ABB RAPID module: P810.mod

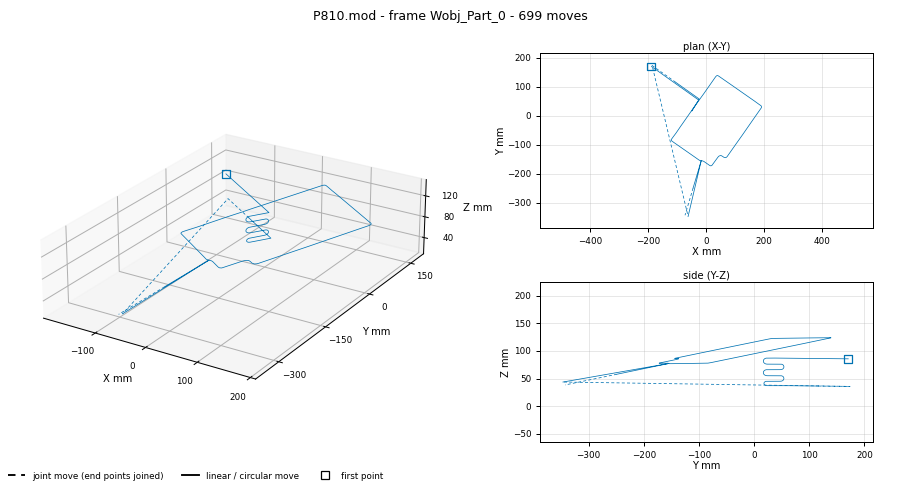
[picture p0: tool path of P810.mod in frame Wobj_Part_0, 699 of 709 moves have a stored position in this frame; points joined in program order, loops and branches not executed]
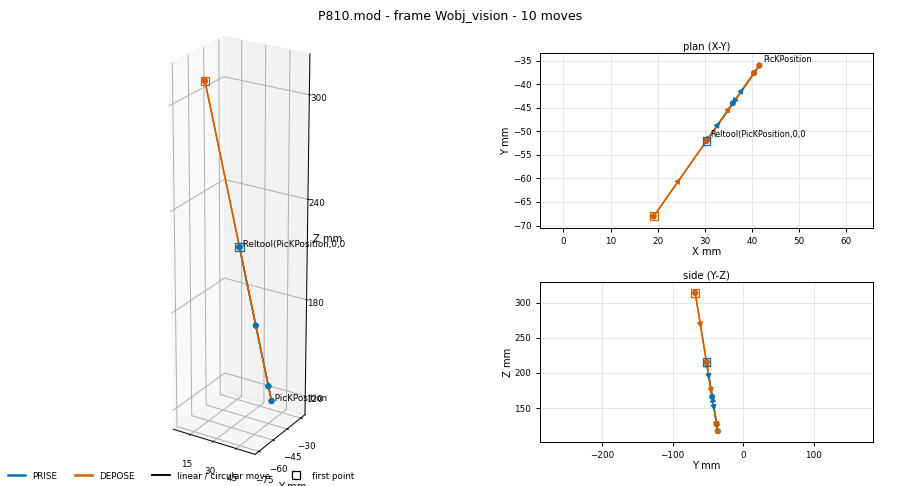
[picture p1: tool path of P810.mod in frame Wobj_vision, 10 of 709 moves have a stored position in this frame; points joined in program order, loops and branches not executed]
MODULE P810

    ! Nom         :P810
    ! Description :
    ! Créé le     :31/05/2023 17:09:28

    LOCAL CONST SPEEDDATA VitesseLente :=[3,500,0,0];
	LOCAL CONST SPEEDDATA VitesseRapide :=[30,500,0,0];
	LOCAL CONST SPEEDDATA VitesseTronconnage :=[2,500,0,0];
	LOCAL CONST SPEEDDATA VitesseTronconnageApp :=[10,500,0,0];
    !
    !Point de prise
    LOCAL PERS Robtarget PicKPosition := [[41.5753348613417,-36.0457521301925,117.430293654676],[0.0866528508359123,-0.450908798340459,0.887153744459286,0.0461602936844953],[0,0,0,0],[8.999999E+09,8.999999E+09,8.999999E+09,8.999999E+09,8.999999E+09,8.999999E+09]];
	LOCAL PERS Pose Ref := [[0,0,0],[1,0,0,0]];
    !
    !Declaration des points de meulage

    !Tr_meulage_motif_1 : Meulage d'un motif
    LOCAL CONST Robtarget Tr_meulage_motif_1_0 := [[-24.86866015625,54.7369140625,87.0190703125],[0.325394831809823,-0.323189731818736,0.626217671016949,-0.630490308557156],[0,0,0,0],[8.999999E+09,8.999999E+09,8.999999E+09,8.999999E+09,8.999999E+09,8.999999E+09]];
    LOCAL CONST Robtarget Tr_meulage_motif_1_1 := [[-25.40796484375,53.8948046875,87.019078125],[0.325394831809823,-0.323189731818736,0.626217671016949,-0.630490308557156],[0,0,0,0],[8.999999E+09,8.999999E+09,8.999999E+09,8.999999E+09,8.999999E+09,8.999999E+09]];
    LOCAL CONST Robtarget Tr_meulage_motif_1_2 := [[-25.94726953125,53.0526953125,87.0190859375],[0.325394831809823,-0.323189731818736,0.626217671016949,-0.630490308557156],[0,0,0,0],[8.999999E+09,8.999999E+09,8.999999E+09,8.999999E+09,8.999999E+09,8.999999E+09]];
    LOCAL CONST Robtarget Tr_meulage_motif_1_3 := [[-26.48657421875,52.2105859375,87.01909375],[0.325394831809823,-0.323189731818736,0.626217671016949,-0.630490308557156],[0,0,0,0],[8.999999E+09,8.999999E+09,8.999999E+09,8.999999E+09,8.999999E+09,8.999999E+09]];
    LOCAL CONST Robtarget Tr_meulage_motif_1_4 := [[-27.025880859375,51.36847265625,87.01909375],[0.325394831809823,-0.323189731818736,0.626217671016949,-0.630490308557156],[0,0,0,0],[8.999999E+09,8.999999E+09,8.999999E+09,8.999999E+09,8.999999E+09,8.999999E+09]];
    LOCAL CONST Robtarget Tr_meulage_motif_1_5 := [[-27.565185546875,50.52636328125,87.0191015625],[0.325394831809823,-0.323189731818736,0.626217671016949,-0.630490308557156],[0,0,0,0],[8.999999E+09,8.999999E+09,8.999999E+09,8.999999E+09,8.999999E+09,8.999999E+09]];
    LOCAL CONST Robtarget Tr_meulage_motif_1_6 := [[-28.104490234375,49.68425390625,87.019109375],[0.325394831809823,-0.323189731818736,0.626217671016949,-0.630490308557156],[0,0,0,0],[8.999999E+09,8.999999E+09,8.999999E+09,8.999999E+09,8.999999E+09,8.999999E+09]];
    LOCAL CONST Robtarget Tr_meulage_motif_1_7 := [[-28.643794921875,48.842140625,87.0191171875],[0.325394831809823,-0.323189731818736,0.626217671016949,-0.630490308557156],[0,0,0,0],[8.999999E+09,8.999999E+09,8.999999E+09,8.999999E+09,8.999999E+09,8.999999E+09]];
    LOCAL CONST Robtarget Tr_meulage_motif_1_8 := [[-29.183099609375,48.00003125,87.019125],[0.325394831809823,-0.323189731818736,0.626217671016949,-0.630490308557156],[0,0,0,0],[8.999999E+09,8.999999E+09,8.999999E+09,8.999999E+09,8.999999E+09,8.999999E+09]];
    LOCAL CONST Robtarget Tr_meulage_motif_1_9 := [[-29.722404296875,47.157921875,87.019125],[0.325394831809823,-0.323189731818736,0.626217671016949,-0.630490308557156],[0,0,0,0],[8.999999E+09,8.999999E+09,8.999999E+09,8.999999E+09,8.999999E+09,8.999999E+09]];
    LOCAL CONST Robtarget Tr_meulage_motif_1_10 := [[-30.2617109375,46.3158125,87.0191328125],[0.325394831809823,-0.323189731818736,0.626217671016949,-0.630490308557156],[0,0,0,0],[8.999999E+09,8.999999E+09,8.999999E+09,8.999999E+09,8.999999E+09,8.999999E+09]];
    LOCAL CONST Robtarget Tr_meulage_motif_1_11 := [[-30.801015625,45.47369921875,87.019140625],[0.325394831809823,-0.323189731818736,0.626217671016949,-0.630490308557156],[0,0,0,0],[8.999999E+09,8.999999E+09,8.999999E+09,8.999999E+09,8.999999E+09,8.999999E+09]];
    LOCAL CONST Robtarget Tr_meulage_motif_1_12 := [[-31.3403203125,44.63158984375,87.0191484375],[0.325394831809823,-0.323189731818736,0.626217671016949,-0.630490308557156],[0,0,0,0],[8.999999E+09,8.999999E+09,8.999999E+09,8.999999E+09,8.999999E+09,8.999999E+09]];
    LOCAL CONST Robtarget Tr_meulage_motif_1_13 := [[-31.879625,43.78948046875,87.01915625],[0.325394831809823,-0.323189731818736,0.626217671016949,-0.630490308557156],[0,0,0,0],[8.999999E+09,8.999999E+09,8.999999E+09,8.999999E+09,8.999999E+09,8.999999E+09]];
    LOCAL CONST Robtarget Tr_meulage_motif_1_14 := [[-32.4189296875,42.9473671875,87.01915625],[0.325394831809823,-0.323189731818736,0.626217671016949,-0.630490308557156],[0,0,0,0],[8.999999E+09,8.999999E+09,8.999999E+09,8.999999E+09,8.999999E+09,8.999999E+09]];
    LOCAL CONST Robtarget Tr_meulage_motif_1_15 := [[-32.958234375,42.1052578125,87.0191640625],[0.325394831809823,-0.323189731818736,0.626217671016949,-0.630490308557156],[0,0,0,0],[8.999999E+09,8.999999E+09,8.999999E+09,8.999999E+09,8.999999E+09,8.999999E+09]];
    LOCAL CONST Robtarget Tr_meulage_motif_1_16 := [[-33.4975390625,41.2631484375,87.019171875],[0.325394831809823,-0.323189731818736,0.626217671016949,-0.630490308557156],[0,0,0,0],[8.999999E+09,8.999999E+09,8.999999E+09,8.999999E+09,8.999999E+09,8.999999E+09]];
    LOCAL CONST Robtarget Tr_meulage_motif_1_17 := [[-34.03684375,40.42103515625,87.0191796875],[0.325394831809823,-0.323189731818736,0.626217671016949,-0.630490308557156],[0,0,0,0],[8.999999E+09,8.999999E+09,8.999999E+09,8.999999E+09,8.999999E+09,8.999999E+09]];
    LOCAL CONST Robtarget Tr_meulage_motif_1_18 := [[-34.5761484375,39.57892578125,87.0191875],[0.325394831809823,-0.323189731818736,0.626217671016949,-0.630490308557156],[0,0,0,0],[8.999999E+09,8.999999E+09,8.999999E+09,8.999999E+09,8.999999E+09,8.999999E+09]];
    LOCAL CONST Robtarget Tr_meulage_motif_1_19 := [[-35.11545703125,38.73681640625,87.0191875],[0.325394831809823,-0.323189731818736,0.626217671016949,-0.630490308557156],[0,0,0,0],[8.999999E+09,8.999999E+09,8.999999E+09,8.999999E+09,8.999999E+09,8.999999E+09]];
    LOCAL CONST Robtarget Tr_meulage_motif_1_20 := [[-35.65476171875,37.89470703125,87.0191953125],[0.325394831809823,-0.323189731818736,0.626217671016949,-0.630490308557156],[0,0,0,0],[8.999999E+09,8.999999E+09,8.999999E+09,8.999999E+09,8.999999E+09,8.999999E+09]];
    LOCAL CONST Robtarget Tr_meulage_motif_1_21 := [[-36.19406640625,37.05259375,87.019203125],[0.325394831809823,-0.323189731818736,0.626217671016949,-0.630490308557156],[0,0,0,0],[8.999999E+09,8.999999E+09,8.999999E+09,8.999999E+09,8.999999E+09,8.999999E+09]];
    LOCAL CONST Robtarget Tr_meulage_motif_1_22 := [[-36.73337109375,36.210484375,87.0192109375],[0.325394831809823,-0.323189731818736,0.626217671016949,-0.630490308557156],[0,0,0,0],[8.999999E+09,8.999999E+09,8.999999E+09,8.999999E+09,8.999999E+09,8.999999E+09]];
    LOCAL CONST Robtarget Tr_meulage_motif_1_23 := [[-37.27267578125,35.368375,87.01921875],[0.325394831809823,-0.323189731818736,0.626217671016949,-0.630490308557156],[0,0,0,0],[8.999999E+09,8.999999E+09,8.999999E+09,8.999999E+09,8.999999E+09,8.999999E+09]];
    LOCAL CONST Robtarget Tr_meulage_motif_1_24 := [[-37.81198046875,34.52626171875,87.0192265625],[0.325394831809823,-0.323189731818736,0.626217671016949,-0.630490308557156],[0,0,0,0],[8.999999E+09,8.999999E+09,8.999999E+09,8.999999E+09,8.999999E+09,8.999999E+09]];
    LOCAL CONST Robtarget Tr_meulage_motif_1_25 := [[-38.35128515625,33.68415234375,87.0192265625],[0.325394831809823,-0.323189731818736,0.626217671016949,-0.630490308557156],[0,0,0,0],[8.999999E+09,8.999999E+09,8.999999E+09,8.999999E+09,8.999999E+09,8.999999E+09]];
    LOCAL CONST Robtarget Tr_meulage_motif_1_26 := [[-38.89058984375,32.84204296875,87.019234375],[0.325394831809823,-0.323189731818736,0.626217671016949,-0.630490308557156],[0,0,0,0],[8.999999E+09,8.999999E+09,8.999999E+09,8.999999E+09,8.999999E+09,8.999999E+09]];
    LOCAL CONST Robtarget Tr_meulage_motif_1_27 := [[-39.42989453125,31.999931640625,87.0192421875],[0.325394831809823,-0.323189731818736,0.626217671016949,-0.630490308557156],[0,0,0,0],[8.999999E+09,8.999999E+09,8.999999E+09,8.999999E+09,8.999999E+09,8.999999E+09]];
    LOCAL CONST Robtarget Tr_meulage_motif_1_28 := [[-39.96919921875,31.157822265625,87.01925],[0.325394831809823,-0.323189731818736,0.626217671016949,-0.630490308557156],[0,0,0,0],[8.999999E+09,8.999999E+09,8.999999E+09,8.999999E+09,8.999999E+09,8.999999E+09]];
    LOCAL CONST Robtarget Tr_meulage_motif_1_29 := [[-40.50850390625,30.3157109375,87.0192578125],[0.325394831809823,-0.323189731818736,0.626217671016949,-0.630490308557156],[0,0,0,0],[8.999999E+09,8.999999E+09,8.999999E+09,8.999999E+09,8.999999E+09,8.999999E+09]];
    LOCAL CONST Robtarget Tr_meulage_motif_1_30 := [[-41.04780859375,29.473599609375,87.0192578125],[0.325394831809823,-0.323189731818736,0.626217671016949,-0.630490308557156],[0,0,0,0],[8.999999E+09,8.999999E+09,8.999999E+09,8.999999E+09,8.999999E+09,8.999999E+09]];
    LOCAL CONST Robtarget Tr_meulage_motif_1_31 := [[-41.58711328125,28.631490234375,87.019265625],[0.325394831809823,-0.323189731818736,0.626217671016949,-0.630490308557156],[0,0,0,0],[8.999999E+09,8.999999E+09,8.999999E+09,8.999999E+09,8.999999E+09,8.999999E+09]];
    LOCAL CONST Robtarget Tr_meulage_motif_1_32 := [[-42.126421875,27.78937890625,87.0192734375],[0.325394831809823,-0.323189731818736,0.626217671016949,-0.630490308557156],[0,0,0,0],[8.999999E+09,8.999999E+09,8.999999E+09,8.999999E+09,8.999999E+09,8.999999E+09]];
    LOCAL CONST Robtarget Tr_meulage_motif_1_33 := [[-42.6657265625,26.94726953125,87.01928125],[0.325394831809823,-0.323189731818736,0.626217671016949,-0.630490308557156],[0,0,0,0],[8.999999E+09,8.999999E+09,8.999999E+09,8.999999E+09,8.999999E+09,8.999999E+09]];
    LOCAL CONST Robtarget Tr_meulage_motif_1_34 := [[-43.20503125,26.105158203125,87.0192890625],[0.325394831809823,-0.323189731818736,0.626217671016949,-0.630490308557156],[0,0,0,0],[8.999999E+09,8.999999E+09,8.999999E+09,8.999999E+09,8.999999E+09,8.999999E+09]];
    LOCAL CONST Robtarget Tr_meulage_motif_1_35 := [[-43.7443359375,25.263046875,87.0192890625],[0.325394831809823,-0.323189731818736,0.626217671016949,-0.630490308557156],[0,0,0,0],[8.999999E+09,8.999999E+09,8.999999E+09,8.999999E+09,8.999999E+09,8.999999E+09]];
    LOCAL CONST Robtarget Tr_meulage_motif_1_36 := [[-44.283640625,24.4209375,87.019296875],[0.325394831809823,-0.323189731818736,0.626217671016949,-0.630490308557156],[0,0,0,0],[8.999999E+09,8.999999E+09,8.999999E+09,8.999999E+09,8.999999E+09,8.999999E+09]];
    LOCAL CONST Robtarget Tr_meulage_motif_1_37 := [[-44.8229453125,23.578826171875,87.0193046875],[0.325394831809823,-0.323189731818736,0.626217671016949,-0.630490308557156],[0,0,0,0],[8.999999E+09,8.999999E+09,8.999999E+09,8.999999E+09,8.999999E+09,8.999999E+09]];
    LOCAL CONST Robtarget Tr_meulage_motif_1_38 := [[-45.36225,22.736716796875,87.0193125],[0.325394831809823,-0.323189731818736,0.626217671016949,-0.630490308557156],[0,0,0,0],[8.999999E+09,8.999999E+09,8.999999E+09,8.999999E+09,8.999999E+09,8.999999E+09]];
    LOCAL CONST Robtarget Tr_meulage_motif_1_39 := [[-45.8972109375,21.90065625,86.9087265625],[0.325394831809823,-0.323189731818736,0.626217671016949,-0.630490308557156],[0,0,0,0],[8.999999E+09,8.999999E+09,8.999999E+09,8.999999E+09,8.999999E+09,8.999999E+09]];
    LOCAL CONST Robtarget Tr_meulage_motif_1_40 := [[-46.40703125,21.10319140625,86.697546875],[0.325394831809823,-0.323189731818736,0.626217671016949,-0.630490308557156],[0,0,0,0],[8.999999E+09,8.999999E+09,8.999999E+09,8.999999E+09,8.999999E+09,8.999999E+09]];
    LOCAL CONST Robtarget Tr_meulage_motif_1_41 := [[-46.86609375,20.384583984375,86.4257109375],[0.325394831809823,-0.323189731818736,0.626217671016949,-0.630490308557156],[0,0,0,0],[8.999999E+09,8.999999E+09,8.999999E+09,8.999999E+09,8.999999E+09,8.999999E+09]];
    LOCAL CONST Robtarget Tr_meulage_motif_1_42 := [[-47.2697109375,19.7525234375,86.1497734375],[0.325394831809823,-0.323189731818736,0.626217671016949,-0.630490308557156],[0,0,0,0],[8.999999E+09,8.999999E+09,8.999999E+09,8.999999E+09,8.999999E+09,8.999999E+09]];
    LOCAL CONST Robtarget Tr_meulage_motif_1_43 := [[-47.861671875,18.824119140625,85.5336640625],[0.325394831809823,-0.323189731818736,0.626217671016949,-0.630490308557156],[0,0,0,0],[8.999999E+09,8.999999E+09,8.999999E+09,8.999999E+09,8.999999E+09,8.999999E+09]];
    LOCAL CONST Robtarget Tr_meulage_motif_1_44 := [[-48.41131640625,17.960271484375,84.686015625],[0.325394831809823,-0.323189731818736,0.626217671016949,-0.630490308557156],[0,0,0,0],[8.999999E+09,8.999999E+09,8.999999E+09,8.999999E+09,8.999999E+09,8.999999E+09]];
    LOCAL CONST Robtarget Tr_meulage_motif_1_45 := [[-48.865390625,17.244478515625,83.66215625],[0.325394831809823,-0.323189731818736,0.626217671016949,-0.630490308557156],[0,0,0,0],[8.999999E+09,8.999999E+09,8.999999E+09,8.999999E+09,8.999999E+09,8.999999E+09]];
    LOCAL CONST Robtarget Tr_meulage_motif_1_46 := [[-49.1253125,16.83124609375,82.5459765625],[0.325394831809823,-0.323189731818736,0.626217671016949,-0.630490308557156],[0,0,0,0],[8.999999E+09,8.999999E+09,8.999999E+09,8.999999E+09,8.999999E+09,8.999999E+09]];
    LOCAL CONST Robtarget Tr_meulage_motif_1_47 := [[-49.13782421875,16.807115234375,81.850015625],[0.325394831809823,-0.323189731818736,0.626217671016949,-0.630490308557156],[0,0,0,0],[8.999999E+09,8.999999E+09,8.999999E+09,8.999999E+09,8.999999E+09,8.999999E+09]];
    LOCAL CONST Robtarget Tr_meulage_motif_1_48 := [[-49.13583984375,16.805841796875,81.188765625],[0.325394831809823,-0.323189731818736,0.626217671016949,-0.630490308557156],[0,0,0,0],[8.999999E+09,8.999999E+09,8.999999E+09,8.999999E+09,8.999999E+09,8.999999E+09]];
    LOCAL CONST Robtarget Tr_meulage_motif_1_49 := [[-49.104265625,16.850779296875,80.5276796875],[0.325394831809823,-0.323189731818736,0.626217671016949,-0.630490308557156],[0,0,0,0],[8.999999E+09,8.999999E+09,8.999999E+09,8.999999E+09,8.999999E+09,8.999999E+09]];
    LOCAL CONST Robtarget Tr_meulage_motif_1_50 := [[-48.8322734375,17.268212890625,79.4259296875],[0.325394831809823,-0.323189731818736,0.626217671016949,-0.630490308557156],[0,0,0,0],[8.999999E+09,8.999999E+09,8.999999E+09,8.999999E+09,8.999999E+09,8.999999E+09]];
    LOCAL CONST Robtarget Tr_meulage_motif_1_51 := [[-48.3672734375,17.987646484375,78.4193046875],[0.325394831809823,-0.323189731818736,0.626217671016949,-0.630490308557156],[0,0,0,0],[8.999999E+09,8.999999E+09,8.999999E+09,8.999999E+09,8.999999E+09,8.999999E+09]];
    LOCAL CONST Robtarget Tr_meulage_motif_1_52 := [[-47.81286328125,18.84787109375,77.5904296875],[0.325394831809823,-0.323189731818736,0.626217671016949,-0.630490308557156],[0,0,0,0],[8.999999E+09,8.999999E+09,8.999999E+09,8.999999E+09,8.999999E+09,8.999999E+09]];
    LOCAL CONST Robtarget Tr_meulage_motif_1_53 := [[-47.441125,19.425716796875,77.1946796875],[0.325394831809823,-0.323189731818736,0.626217671016949,-0.630490308557156],[0,0,0,0],[8.999999E+09,8.999999E+09,8.999999E+09,8.999999E+09,8.999999E+09,8.999999E+09]];
    LOCAL CONST Robtarget Tr_meulage_motif_1_54 := [[-46.8150625,20.40007421875,76.707140625],[0.325394831809823,-0.323189731818736,0.626217671016949,-0.630490308557156],[0,0,0,0],[8.999999E+09,8.999999E+09,8.999999E+09,8.999999E+09,8.999999E+09,8.999999E+09]];
    LOCAL CONST Robtarget Tr_meulage_motif_1_55 := [[-46.35854296875,21.111173828125,76.443046875],[0.325394831809823,-0.323189731818736,0.626217671016949,-0.630490308557156],[0,0,0,0],[8.999999E+09,8.999999E+09,8.999999E+09,8.999999E+09,8.999999E+09,8.999999E+09]];
    LOCAL CONST Robtarget Tr_meulage_motif_1_56 := [[-45.855296875,21.895626953125,76.2385703125],[0.325394831809823,-0.323189731818736,0.626217671016949,-0.630490308557156],[0,0,0,0],[8.999999E+09,8.999999E+09,8.999999E+09,8.999999E+09,8.999999E+09,8.999999E+09]];
    LOCAL CONST Robtarget Tr_meulage_motif_1_57 := [[-45.32561328125,22.722001953125,76.1299765625],[0.325394831809823,-0.323189731818736,0.626217671016949,-0.630490308557156],[0,0,0,0],[8.999999E+09,8.999999E+09,8.999999E+09,8.999999E+09,8.999999E+09,8.999999E+09]];
    LOCAL CONST Robtarget Tr_meulage_motif_1_58 := [[-44.789984375,23.55763671875,76.019375],[0.325394831809823,-0.323189731818736,0.626217671016949,-0.630490308557156],[0,0,0,0],[8.999999E+09,8.999999E+09,8.999999E+09,8.999999E+09,8.999999E+09,8.999999E+09]];
    LOCAL CONST Robtarget Tr_meulage_motif_1_59 := [[-44.2506796875,24.399748046875,76.0193671875],[0.325394831809823,-0.323189731818736,0.626217671016949,-0.630490308557156],[0,0,0,0],[8.999999E+09,8.999999E+09,8.999999E+09,8.999999E+09,8.999999E+09,8.999999E+09]];
    LOCAL CONST Robtarget Tr_meulage_motif_1_60 := [[-43.711375,25.241857421875,76.019359375],[0.325394831809823,-0.323189731818736,0.626217671016949,-0.630490308557156],[0,0,0,0],[8.999999E+09,8.999999E+09,8.999999E+09,8.999999E+09,8.999999E+09,8.999999E+09]];
    LOCAL CONST Robtarget Tr_meulage_motif_1_61 := [[-43.1720703125,26.08396875,76.019359375],[0.325394831809823,-0.323189731818736,0.626217671016949,-0.630490308557156],[0,0,0,0],[8.999999E+09,8.999999E+09,8.999999E+09,8.999999E+09,8.999999E+09,8.999999E+09]];
    LOCAL CONST Robtarget Tr_meulage_motif_1_62 := [[-42.632765625,26.926078125,76.0193515625],[0.325394831809823,-0.323189731818736,0.626217671016949,-0.630490308557156],[0,0,0,0],[8.999999E+09,8.999999E+09,8.999999E+09,8.999999E+09,8.999999E+09,8.999999E+09]];
    LOCAL CONST Robtarget Tr_meulage_motif_1_63 := [[-42.0934609375,27.768189453125,76.01934375],[0.325394831809823,-0.323189731818736,0.626217671016949,-0.630490308557156],[0,0,0,0],[8.999999E+09,8.999999E+09,8.999999E+09,8.999999E+09,8.999999E+09,8.999999E+09]];
    LOCAL CONST Robtarget Tr_meulage_motif_1_64 := [[-41.55415625,28.61030078125,76.0193359375],[0.325394831809823,-0.323189731818736,0.626217671016949,-0.630490308557156],[0,0,0,0],[8.999999E+09,8.999999E+09,8.999999E+09,8.999999E+09,8.999999E+09,8.999999E+09]];
    LOCAL CONST Robtarget Tr_meulage_motif_1_65 := [[-41.0148515625,29.45241015625,76.019328125],[0.325394831809823,-0.323189731818736,0.626217671016949,-0.630490308557156],[0,0,0,0],[8.999999E+09,8.999999E+09,8.999999E+09,8.999999E+09,8.999999E+09,8.999999E+09]];
    LOCAL CONST Robtarget Tr_meulage_motif_1_66 := [[-40.475546875,30.294521484375,76.0193203125],[0.325394831809823,-0.323189731818736,0.626217671016949,-0.630490308557156],[0,0,0,0],[8.999999E+09,8.999999E+09,8.999999E+09,8.999999E+09,8.999999E+09,8.999999E+09]];
    LOCAL CONST Robtarget Tr_meulage_motif_1_67 := [[-39.9362421875,31.136630859375,76.0193203125],[0.325394831809823,-0.323189731818736,0.626217671016949,-0.630490308557156],[0,0,0,0],[8.999999E+09,8.999999E+09,8.999999E+09,8.999999E+09,8.999999E+09,8.999999E+09]];
    LOCAL CONST Robtarget Tr_meulage_motif_1_68 := [[-39.3969375,31.9787421875,76.0193125],[0.325394831809823,-0.323189731818736,0.626217671016949,-0.630490308557156],[0,0,0,0],[8.999999E+09,8.999999E+09,8.999999E+09,8.999999E+09,8.999999E+09,8.999999E+09]];
    LOCAL CONST Robtarget Tr_meulage_motif_1_69 := [[-38.8576328125,32.8208515625,76.0193046875],[0.325394831809823,-0.323189731818736,0.626217671016949,-0.630490308557156],[0,0,0,0],[8.999999E+09,8.999999E+09,8.999999E+09,8.999999E+09,8.999999E+09,8.999999E+09]];
    LOCAL CONST Robtarget Tr_meulage_motif_1_70 := [[-38.318328125,33.66296484375,76.019296875],[0.325394831809823,-0.323189731818736,0.626217671016949,-0.630490308557156],[0,0,0,0],[8.999999E+09,8.999999E+09,8.999999E+09,8.999999E+09,8.999999E+09,8.999999E+09]];
    LOCAL CONST Robtarget Tr_meulage_motif_1_71 := [[-37.77901953125,34.50507421875,76.0192890625],[0.325394831809823,-0.323189731818736,0.626217671016949,-0.630490308557156],[0,0,0,0],[8.999999E+09,8.999999E+09,8.999999E+09,8.999999E+09,8.999999E+09,8.999999E+09]];
    LOCAL CONST Robtarget Tr_meulage_motif_1_72 := [[-37.23971484375,35.34718359375,76.0192890625],[0.325394831809823,-0.323189731818736,0.626217671016949,-0.630490308557156],[0,0,0,0],[8.999999E+09,8.999999E+09,8.999999E+09,8.999999E+09,8.999999E+09,8.999999E+09]];
    LOCAL CONST Robtarget Tr_meulage_motif_1_73 := [[-36.70041015625,36.18929296875,76.01928125],[0.325394831809823,-0.323189731818736,0.626217671016949,-0.630490308557156],[0,0,0,0],[8.999999E+09,8.999999E+09,8.999999E+09,8.999999E+09,8.999999E+09,8.999999E+09]];
    LOCAL CONST Robtarget Tr_meulage_motif_1_74 := [[-36.16110546875,37.03140625,76.0192734375],[0.325394831809823,-0.323189731818736,0.626217671016949,-0.630490308557156],[0,0,0,0],[8.999999E+09,8.999999E+09,8.999999E+09,8.999999E+09,8.999999E+09,8.999999E+09]];
    LOCAL CONST Robtarget Tr_meulage_motif_1_75 := [[-35.62180078125,37.873515625,76.019265625],[0.325394831809823,-0.323189731818736,0.626217671016949,-0.630490308557156],[0,0,0,0],[8.999999E+09,8.999999E+09,8.999999E+09,8.999999E+09,8.999999E+09,8.999999E+09]];
    LOCAL CONST Robtarget Tr_meulage_motif_1_76 := [[-35.08249609375,38.715625,76.0192578125],[0.325394831809823,-0.323189731818736,0.626217671016949,-0.630490308557156],[0,0,0,0],[8.999999E+09,8.999999E+09,8.999999E+09,8.999999E+09,8.999999E+09,8.999999E+09]];
    LOCAL CONST Robtarget Tr_meulage_motif_1_77 := [[-34.54319140625,39.55773828125,76.0192578125],[0.325394831809823,-0.323189731818736,0.626217671016949,-0.630490308557156],[0,0,0,0],[8.999999E+09,8.999999E+09,8.999999E+09,8.999999E+09,8.999999E+09,8.999999E+09]];
    LOCAL CONST Robtarget Tr_meulage_motif_1_78 := [[-34.00388671875,40.39984765625,76.01925],[0.325394831809823,-0.323189731818736,0.626217671016949,-0.630490308557156],[0,0,0,0],[8.999999E+09,8.999999E+09,8.999999E+09,8.999999E+09,8.999999E+09,8.999999E+09]];
    LOCAL CONST Robtarget Tr_meulage_motif_1_79 := [[-33.46458203125,41.24195703125,76.0192421875],[0.325394831809823,-0.323189731818736,0.626217671016949,-0.630490308557156],[0,0,0,0],[8.999999E+09,8.999999E+09,8.999999E+09,8.999999E+09,8.999999E+09,8.999999E+09]];
    LOCAL CONST Robtarget Tr_meulage_motif_1_80 := [[-32.92527734375,42.08406640625,76.019234375],[0.325394831809823,-0.323189731818736,0.626217671016949,-0.630490308557156],[0,0,0,0],[8.999999E+09,8.999999E+09,8.999999E+09,8.999999E+09,8.999999E+09,8.999999E+09]];
    LOCAL CONST Robtarget Tr_meulage_motif_1_81 := [[-32.385970703125,42.9261796875,76.0192265625],[0.325394831809823,-0.323189731818736,0.626217671016949,-0.630490308557156],[0,0,0,0],[8.999999E+09,8.999999E+09,8.999999E+09,8.999999E+09,8.999999E+09,8.999999E+09]];
    LOCAL CONST Robtarget Tr_meulage_motif_1_82 := [[-31.846666015625,43.7682890625,76.0192265625],[0.325394831809823,-0.323189731818736,0.626217671016949,-0.630490308557156],[0,0,0,0],[8.999999E+09,8.999999E+09,8.999999E+09,8.999999E+09,8.999999E+09,8.999999E+09]];
    LOCAL CONST Robtarget Tr_meulage_motif_1_83 := [[-31.307361328125,44.6103984375,76.01921875],[0.325394831809823,-0.323189731818736,0.626217671016949,-0.630490308557156],[0,0,0,0],[8.999999E+09,8.999999E+09,8.999999E+09,8.999999E+09,8.999999E+09,8.999999E+09]];
    LOCAL CONST Robtarget Tr_meulage_motif_1_84 := [[-30.768056640625,45.45251171875,76.0192109375],[0.325394831809823,-0.323189731818736,0.626217671016949,-0.630490308557156],[0,0,0,0],[8.999999E+09,8.999999E+09,8.999999E+09,8.999999E+09,8.999999E+09,8.999999E+09]];
    LOCAL CONST Robtarget Tr_meulage_motif_1_85 := [[-30.228751953125,46.29462109375,76.019203125],[0.325394831809823,-0.323189731818736,0.626217671016949,-0.630490308557156],[0,0,0,0],[8.999999E+09,8.999999E+09,8.999999E+09,8.999999E+09,8.999999E+09,8.999999E+09]];
    LOCAL CONST Robtarget Tr_meulage_motif_1_86 := [[-29.689447265625,47.13673046875,76.0191953125],[0.325394831809823,-0.323189731818736,0.626217671016949,-0.630490308557156],[0,0,0,0],[8.999999E+09,8.999999E+09,8.999999E+09,8.999999E+09,8.999999E+09,8.999999E+09]];
    LOCAL CONST Robtarget Tr_meulage_motif_1_87 := [[-29.150140625,47.97884375,76.0191953125],[0.325394831809823,-0.323189731818736,0.626217671016949,-0.630490308557156],[0,0,0,0],[8.999999E+09,8.999999E+09,8.999999E+09,8.999999E+09,8.999999E+09,8.999999E+09]];
    LOCAL CONST Robtarget Tr_meulage_motif_1_88 := [[-28.6108359375,48.820953125,76.0191875],[0.325394831809823,-0.323189731818736,0.626217671016949,-0.630490308557156],[0,0,0,0],[8.999999E+09,8.999999E+09,8.999999E+09,8.999999E+09,8.999999E+09,8.999999E+09]];
    LOCAL CONST Robtarget Tr_meulage_motif_1_89 := [[-28.0752109375,49.6565859375,75.9085859375],[0.325394831809823,-0.323189731818736,0.626217671016949,-0.630490308557156],[0,0,0,0],[8.999999E+09,8.999999E+09,8.999999E+09,8.999999E+09,8.999999E+09,8.999999E+09]];
    LOCAL CONST Robtarget Tr_meulage_motif_1_90 := [[-27.564126953125,50.45323828125,75.697390625],[0.325394831809823,-0.323189731818736,0.626217671016949,-0.630490308557156],[0,0,0,0],[8.999999E+09,8.999999E+09,8.999999E+09,8.999999E+09,8.999999E+09,8.999999E+09]];
    LOCAL CONST Robtarget Tr_meulage_motif_1_91 := [[-27.103435546875,51.170796875,75.425546875],[0.325394831809823,-0.323189731818736,0.626217671016949,-0.630490308557156],[0,0,0,0],[8.999999E+09,8.999999E+09,8.999999E+09,8.999999E+09,8.999999E+09,8.999999E+09]];
    LOCAL CONST Robtarget Tr_meulage_motif_1_92 := [[-26.71880859375,51.76937109375,75.121390625],[0.325394831809823,-0.323189731818736,0.626217671016949,-0.630490308557156],[0,0,0,0],[8.999999E+09,8.999999E+09,8.999999E+09,8.999999E+09,8.999999E+09,8.999999E+09]];
    LOCAL CONST Robtarget Tr_meulage_motif_1_93 := [[-26.1589296875,52.639234375,74.4588515625],[0.325394831809823,-0.323189731818736,0.626217671016949,-0.630490308557156],[0,0,0,0],[8.999999E+09,8.999999E+09,8.999999E+09,8.999999E+09,8.999999E+09,8.999999E+09]];
    LOCAL CONST Robtarget Tr_meulage_motif_1_94 := [[-25.66980859375,53.39702734375,73.5569140625],[0.325394831809823,-0.323189731818736,0.626217671016949,-0.630490308557156],[0,0,0,0],[8.999999E+09,8.999999E+09,8.999999E+09,8.999999E+09,8.999999E+09,8.999999E+09]];
    LOCAL CONST Robtarget Tr_meulage_motif_1_95 := [[-25.378162109375,53.845515625,72.510890625],[0.325394831809823,-0.323189731818736,0.626217671016949,-0.630490308557156],[0,0,0,0],[8.999999E+09,8.999999E+09,8.999999E+09,8.999999E+09,8.999999E+09,8.999999E+09]];
    LOCAL CONST Robtarget Tr_meulage_motif_1_96 := [[-25.276431640625,53.99978515625,71.817671875],[0.325394831809823,-0.323189731818736,0.626217671016949,-0.630490308557156],[0,0,0,0],[8.999999E+09,8.999999E+09,8.999999E+09,8.999999E+09,8.999999E+09,8.999999E+09]];
    LOCAL CONST Robtarget Tr_meulage_motif_1_97 := [[-25.239693359375,54.05206640625,71.0476796875],[0.325394831809823,-0.323189731818736,0.626217671016949,-0.630490308557156],[0,0,0,0],[8.999999E+09,8.999999E+09,8.999999E+09,8.999999E+09,8.999999E+09,8.999999E+09]];
    LOCAL CONST Robtarget Tr_meulage_motif_1_98 := [[-25.273486328125,53.99421484375,70.2778046875],[0.325394831809823,-0.323189731818736,0.626217671016949,-0.630490308557156],[0,0,0,0],[8.999999E+09,8.999999E+09,8.999999E+09,8.999999E+09,8.999999E+09,8.999999E+09]];
    LOCAL CONST Robtarget Tr_meulage_motif_1_99 := [[-25.496455078125,53.638734375,69.1695703125],[0.325394831809823,-0.323189731818736,0.626217671016949,-0.630490308557156],[0,0,0,0],[8.999999E+09,8.999999E+09,8.999999E+09,8.999999E+09,8.999999E+09,8.999999E+09]];
    LOCAL CONST Robtarget Tr_meulage_motif_1_100 := [[-25.718140625,53.2887109375,68.5838828125],[0.325394831809823,-0.323189731818736,0.626217671016949,-0.630490308557156],[0,0,0,0],[8.999999E+09,8.999999E+09,8.999999E+09,8.999999E+09,8.999999E+09,8.999999E+09]];
    LOCAL CONST Robtarget Tr_meulage_motif_1_101 := [[-26.1939140625,52.5399453125,67.6967734375],[0.325394831809823,-0.323189731818736,0.626217671016949,-0.630490308557156],[0,0,0,0],[8.999999E+09,8.999999E+09,8.999999E+09,8.999999E+09,8.999999E+09,8.999999E+09]];
    LOCAL CONST Robtarget Tr_meulage_motif_1_102 := [[-26.508537109375,52.04593359375,67.28246875],[0.325394831809823,-0.323189731818736,0.626217671016949,-0.630490308557156],[0,0,0,0],[8.999999E+09,8.999999E+09,8.999999E+09,8.999999E+09,8.999999E+09,8.999999E+09]];
    LOCAL CONST Robtarget Tr_meulage_motif_1_103 := [[-27.109798828125,51.103484375,66.7383828125],[0.325394831809823,-0.323189731818736,0.626217671016949,-0.630490308557156],[0,0,0,0],[8.999999E+09,8.999999E+09,8.999999E+09,8.999999E+09,8.999999E+09,8.999999E+09]];
    LOCAL CONST Robtarget Tr_meulage_motif_1_104 := [[-27.55416015625,50.407671875,66.442890625],[0.325394831809823,-0.323189731818736,0.626217671016949,-0.630490308557156],[0,0,0,0],[8.999999E+09,8.999999E+09,8.999999E+09,8.999999E+09,8.999999E+09,8.999999E+09]];
    LOCAL CONST Robtarget Tr_meulage_motif_1_105 := [[-28.0561796875,49.62243359375,66.2384296875],[0.325394831809823,-0.323189731818736,0.626217671016949,-0.630490308557156],[0,0,0,0],[8.999999E+09,8.999999E+09,8.999999E+09,8.999999E+09,8.999999E+09,8.999999E+09]];
    LOCAL CONST Robtarget Tr_meulage_motif_1_106 := [[-28.585216796875,48.79563671875,66.12984375],[0.325394831809823,-0.323189731818736,0.626217671016949,-0.630490308557156],[0,0,0,0],[8.999999E+09,8.999999E+09,8.999999E+09,8.999999E+09,8.999999E+09,8.999999E+09]];
    LOCAL CONST Robtarget Tr_meulage_motif_1_107 := [[-29.1201796875,47.959578125,66.0192578125],[0.325394831809823,-0.323189731818736,0.626217671016949,-0.630490308557156],[0,0,0,0],[8.999999E+09,8.999999E+09,8.999999E+09,8.999999E+09,8.999999E+09,8.999999E+09]];
    LOCAL CONST Robtarget Tr_meulage_motif_1_108 := [[-29.659484375,47.11746875,66.0192578125],[0.325394831809823,-0.323189731818736,0.626217671016949,-0.630490308557156],[0,0,0,0],[8.999999E+09,8.999999E+09,8.999999E+09,8.999999E+09,8.999999E+09,8.999999E+09]];
    LOCAL CONST Robtarget Tr_meulage_motif_1_109 := [[-30.1987890625,46.27535546875,66.019265625],[0.325394831809823,-0.323189731818736,0.626217671016949,-0.630490308557156],[0,0,0,0],[8.999999E+09,8.999999E+09,8.999999E+09,8.999999E+09,8.999999E+09,8.999999E+09]];
    LOCAL CONST Robtarget Tr_meulage_motif_1_110 := [[-30.73809375,45.43324609375,66.0192734375],[0.325394831809823,-0.323189731818736,0.626217671016949,-0.630490308557156],[0,0,0,0],[8.999999E+09,8.999999E+09,8.999999E+09,8.999999E+09,8.999999E+09,8.999999E+09]];
    LOCAL CONST Robtarget Tr_meulage_motif_1_111 := [[-31.2773984375,44.59113671875,66.01928125],[0.325394831809823,-0.323189731818736,0.626217671016949,-0.630490308557156],[0,0,0,0],[8.999999E+09,8.999999E+09,8.999999E+09,8.999999E+09,8.999999E+09,8.999999E+09]];
    LOCAL CONST Robtarget Tr_meulage_motif_1_112 := [[-31.816703125,43.74902734375,66.0192890625],[0.325394831809823,-0.323189731818736,0.626217671016949,-0.630490308557156],[0,0,0,0],[8.999999E+09,8.999999E+09,8.999999E+09,8.999999E+09,8.999999E+09,8.999999E+09]];
    LOCAL CONST Robtarget Tr_meulage_motif_1_113 := [[-32.3560078125,42.9069140625,66.0192890625],[0.325394831809823,-0.323189731818736,0.626217671016949,-0.630490308557156],[0,0,0,0],[8.999999E+09,8.999999E+09,8.999999E+09,8.999999E+09,8.999999E+09,8.999999E+09]];
    LOCAL CONST Robtarget Tr_meulage_motif_1_114 := [[-32.8953125,42.0648046875,66.019296875],[0.325394831809823,-0.323189731818736,0.626217671016949,-0.630490308557156],[0,0,0,0],[8.999999E+09,8.999999E+09,8.999999E+09,8.999999E+09,8.999999E+09,8.999999E+09]];
    LOCAL CONST Robtarget Tr_meulage_motif_1_115 := [[-33.4346171875,41.2226953125,66.0193046875],[0.325394831809823,-0.323189731818736,0.626217671016949,-0.630490308557156],[0,0,0,0],[8.999999E+09,8.999999E+09,8.999999E+09,8.999999E+09,8.999999E+09,8.999999E+09]];
    LOCAL CONST Robtarget Tr_meulage_motif_1_116 := [[-33.973921875,40.38058203125,66.0193125],[0.325394831809823,-0.323189731818736,0.626217671016949,-0.630490308557156],[0,0,0,0],[8.999999E+09,8.999999E+09,8.999999E+09,8.999999E+09,8.999999E+09,8.999999E+09]];
    LOCAL CONST Robtarget Tr_meulage_motif_1_117 := [[-34.51323046875,39.53847265625,66.0193203125],[0.325394831809823,-0.323189731818736,0.626217671016949,-0.630490308557156],[0,0,0,0],[8.999999E+09,8.999999E+09,8.999999E+09,8.999999E+09,8.999999E+09,8.999999E+09]];
    LOCAL CONST Robtarget Tr_meulage_motif_1_118 := [[-35.05253515625,38.69636328125,66.019328125],[0.325394831809823,-0.323189731818736,0.626217671016949,-0.630490308557156],[0,0,0,0],[8.999999E+09,8.999999E+09,8.999999E+09,8.999999E+09,8.999999E+09,8.999999E+09]];
    LOCAL CONST Robtarget Tr_meulage_motif_1_119 := [[-35.59183984375,37.85425390625,66.019328125],[0.325394831809823,-0.323189731818736,0.626217671016949,-0.630490308557156],[0,0,0,0],[8.999999E+09,8.999999E+09,8.999999E+09,8.999999E+09,8.999999E+09,8.999999E+09]];
    LOCAL CONST Robtarget Tr_meulage_motif_1_120 := [[-36.13114453125,37.012140625,66.0193359375],[0.325394831809823,-0.323189731818736,0.626217671016949,-0.630490308557156],[0,0,0,0],[8.999999E+09,8.999999E+09,8.999999E+09,8.999999E+09,8.999999E+09,8.999999E+09]];
    LOCAL CONST Robtarget Tr_meulage_motif_1_121 := [[-36.67044921875,36.17003125,66.01934375],[0.325394831809823,-0.323189731818736,0.626217671016949,-0.630490308557156],[0,0,0,0],[8.999999E+09,8.999999E+09,8.999999E+09,8.999999E+09,8.999999E+09,8.999999E+09]];
    LOCAL CONST Robtarget Tr_meulage_motif_1_122 := [[-37.20975390625,35.327921875,66.0193515625],[0.325394831809823,-0.323189731818736,0.626217671016949,-0.630490308557156],[0,0,0,0],[8.999999E+09,8.999999E+09,8.999999E+09,8.999999E+09,8.999999E+09,8.999999E+09]];
    LOCAL CONST Robtarget Tr_meulage_motif_1_123 := [[-37.74905859375,34.48580859375,66.019359375],[0.325394831809823,-0.323189731818736,0.626217671016949,-0.630490308557156],[0,0,0,0],[8.999999E+09,8.999999E+09,8.999999E+09,8.999999E+09,8.999999E+09,8.999999E+09]];
    LOCAL CONST Robtarget Tr_meulage_motif_1_124 := [[-38.28836328125,33.64369921875,66.019359375],[0.325394831809823,-0.323189731818736,0.626217671016949,-0.630490308557156],[0,0,0,0],[8.999999E+09,8.999999E+09,8.999999E+09,8.999999E+09,8.999999E+09,8.999999E+09]];
    LOCAL CONST Robtarget Tr_meulage_motif_1_125 := [[-38.82766796875,32.80158984375,66.0193671875],[0.325394831809823,-0.323189731818736,0.626217671016949,-0.630490308557156],[0,0,0,0],[8.999999E+09,8.999999E+09,8.999999E+09,8.999999E+09,8.999999E+09,8.999999E+09]];
    LOCAL CONST Robtarget Tr_meulage_motif_1_126 := [[-39.36697265625,31.959478515625,66.019375],[0.325394831809823,-0.323189731818736,0.626217671016949,-0.630490308557156],[0,0,0,0],[8.999999E+09,8.999999E+09,8.999999E+09,8.999999E+09,8.999999E+09,8.999999E+09]];
    LOCAL CONST Robtarget Tr_meulage_motif_1_127 := [[-39.90627734375,31.1173671875,66.0193828125],[0.325394831809823,-0.323189731818736,0.626217671016949,-0.630490308557156],[0,0,0,0],[8.999999E+09,8.999999E+09,8.999999E+09,8.999999E+09,8.999999E+09,8.999999E+09]];
    LOCAL CONST Robtarget Tr_meulage_motif_1_128 := [[-40.44558203125,30.2752578125,66.019390625],[0.325394831809823,-0.323189731818736,0.626217671016949,-0.630490308557156],[0,0,0,0],[8.999999E+09,8.999999E+09,8.999999E+09,8.999999E+09,8.999999E+09,8.999999E+09]];
    LOCAL CONST Robtarget Tr_meulage_motif_1_129 := [[-40.984890625,29.433146484375,66.019390625],[0.325394831809823,-0.323189731818736,0.626217671016949,-0.630490308557156],[0,0,0,0],[8.999999E+09,8.999999E+09,8.999999E+09,8.999999E+09,8.999999E+09,8.999999E+09]];
    LOCAL CONST Robtarget Tr_meulage_motif_1_130 := [[-41.5241953125,28.591037109375,66.0193984375],[0.325394831809823,-0.323189731818736,0.626217671016949,-0.630490308557156],[0,0,0,0],[8.999999E+09,8.999999E+09,8.999999E+09,8.999999E+09,8.999999E+09,8.999999E+09]];
    LOCAL CONST Robtarget Tr_meulage_motif_1_131 := [[-42.0635,27.74892578125,66.01940625],[0.325394831809823,-0.323189731818736,0.626217671016949,-0.630490308557156],[0,0,0,0],[8.999999E+09,8.999999E+09,8.999999E+09,8.999999E+09,8.999999E+09,8.999999E+09]];
    LOCAL CONST Robtarget Tr_meulage_motif_1_132 := [[-42.6028046875,26.906814453125,66.0194140625],[0.325394831809823,-0.323189731818736,0.626217671016949,-0.630490308557156],[0,0,0,0],[8.999999E+09,8.999999E+09,8.999999E+09,8.999999E+09,8.999999E+09,8.999999E+09]];
    LOCAL CONST Robtarget Tr_meulage_motif_1_133 := [[-43.142109375,26.064705078125,66.019421875],[0.325394831809823,-0.323189731818736,0.626217671016949,-0.630490308557156],[0,0,0,0],[8.999999E+09,8.999999E+09,8.999999E+09,8.999999E+09,8.999999E+09,8.999999E+09]];
    LOCAL CONST Robtarget Tr_meulage_motif_1_134 := [[-43.6814140625,25.22259375,66.019421875],[0.325394831809823,-0.323189731818736,0.626217671016949,-0.630490308557156],[0,0,0,0],[8.999999E+09,8.999999E+09,8.999999E+09,8.999999E+09,8.999999E+09,8.999999E+09]];
    LOCAL CONST Robtarget Tr_meulage_motif_1_135 := [[-44.22071875,24.380484375,66.0194296875],[0.325394831809823,-0.323189731818736,0.626217671016949,-0.630490308557156],[0,0,0,0],[8.999999E+09,8.999999E+09,8.999999E+09,8.999999E+09,8.999999E+09,8.999999E+09]];
    LOCAL CONST Robtarget Tr_meulage_motif_1_136 := [[-44.7600234375,23.538373046875,66.0194375],[0.325394831809823,-0.323189731818736,0.626217671016949,-0.630490308557156],[0,0,0,0],[8.999999E+09,8.999999E+09,8.999999E+09,8.999999E+09,8.999999E+09,8.999999E+09]];
    LOCAL CONST Robtarget Tr_meulage_motif_1_137 := [[-45.299328125,22.696263671875,66.0194453125],[0.325394831809823,-0.323189731818736,0.626217671016949,-0.630490308557156],[0,0,0,0],[8.999999E+09,8.999999E+09,8.999999E+09,8.999999E+09,8.999999E+09,8.999999E+09]];
    LOCAL CONST Robtarget Tr_meulage_motif_1_138 := [[-45.83429296875,21.860203125,65.908859375],[0.325394831809823,-0.323189731818736,0.626217671016949,-0.630490308557156],[0,0,0,0],[8.999999E+09,8.999999E+09,8.999999E+09,8.999999E+09,8.999999E+09,8.999999E+09]];
    LOCAL CONST Robtarget Tr_meulage_motif_1_139 := [[-46.344109375,21.06273828125,65.6976796875],[0.325394831809823,-0.323189731818736,0.626217671016949,-0.630490308557156],[0,0,0,0],[8.999999E+09,8.999999E+09,8.999999E+09,8.999999E+09,8.999999E+09,8.999999E+09]];
    LOCAL CONST Robtarget Tr_meulage_motif_1_140 := [[-46.803171875,20.344130859375,65.42583984375],[0.325394831809823,-0.323189731818736,0.626217671016949,-0.630490308557156],[0,0,0,0],[8.999999E+09,8.999999E+09,8.999999E+09,8.999999E+09,8.999999E+09,8.999999E+09]];
    LOCAL CONST Robtarget Tr_meulage_motif_1_141 := [[-47.2067890625,19.712068359375,65.14991015625],[0.325394831809823,-0.323189731818736,0.626217671016949,-0.630490308557156],[0,0,0,0],[8.999999E+09,8.999999E+09,8.999999E+09,8.999999E+09,8.999999E+09,8.999999E+09]];
    LOCAL CONST Robtarget Tr_meulage_motif_1_142 := [[-47.79875390625,18.783666015625,64.533796875],[0.325394831809823,-0.323189731818736,0.626217671016949,-0.630490308557156],[0,0,0,0],[8.999999E+09,8.999999E+09,8.999999E+09,8.999999E+09,8.999999E+09,8.999999E+09]];
    LOCAL CONST Robtarget Tr_meulage_motif_1_143 := [[-48.34839453125,17.91981640625,63.68615234375],[0.325394831809823,-0.323189731818736,0.626217671016949,-0.630490308557156],[0,0,0,0],[8.999999E+09,8.999999E+09,8.999999E+09,8.999999E+09,8.999999E+09,8.999999E+09]];
    LOCAL CONST Robtarget Tr_meulage_motif_1_144 := [[-48.80247265625,17.204025390625,62.6622890625],[0.325394831809823,-0.323189731818736,0.626217671016949,-0.630490308557156],[0,0,0,0],[8.999999E+09,8.999999E+09,8.999999E+09,8.999999E+09,8.999999E+09,8.999999E+09]];
    LOCAL CONST Robtarget Tr_meulage_motif_1_145 := [[-49.062390625,16.79079296875,61.546109375],[0.325394831809823,-0.323189731818736,0.626217671016949,-0.630490308557156],[0,0,0,0],[8.999999E+09,8.999999E+09,8.999999E+09,8.999999E+09,8.999999E+09,8.999999E+09]];
    LOCAL CONST Robtarget Tr_meulage_motif_1_146 := [[-49.07490234375,16.766662109375,60.85014453125],[0.325394831809823,-0.323189731818736,0.626217671016949,-0.630490308557156],[0,0,0,0],[8.999999E+09,8.999999E+09,8.999999E+09,8.999999E+09,8.999999E+09,8.999999E+09]];
    LOCAL CONST Robtarget Tr_meulage_motif_1_147 := [[-49.072921875,16.765388671875,60.18890234375],[0.325394831809823,-0.323189731818736,0.626217671016949,-0.630490308557156],[0,0,0,0],[8.999999E+09,8.999999E+09,8.999999E+09,8.999999E+09,8.999999E+09,8.999999E+09]];
    LOCAL CONST Robtarget Tr_meulage_motif_1_148 := [[-49.04134375,16.810326171875,59.5278125],[0.325394831809823,-0.323189731818736,0.626217671016949,-0.630490308557156],[0,0,0,0],[8.999999E+09,8.999999E+09,8.999999E+09,8.999999E+09,8.999999E+09,8.999999E+09]];
    LOCAL CONST Robtarget Tr_meulage_motif_1_149 := [[-48.7693515625,17.227759765625,58.42606640625],[0.325394831809823,-0.323189731818736,0.626217671016949,-0.630490308557156],[0,0,0,0],[8.999999E+09,8.999999E+09,8.999999E+09,8.999999E+09,8.999999E+09,8.999999E+09]];
    LOCAL CONST Robtarget Tr_meulage_motif_1_150 := [[-48.30435546875,17.947193359375,57.41944140625],[0.325394831809823,-0.323189731818736,0.626217671016949,-0.630490308557156],[0,0,0,0],[8.999999E+09,8.999999E+09,8.999999E+09,8.999999E+09,8.999999E+09,8.999999E+09]];
    LOCAL CONST Robtarget Tr_meulage_motif_1_151 := [[-47.74994140625,18.80741796875,56.5905625],[0.325394831809823,-0.323189731818736,0.626217671016949,-0.630490308557156],[0,0,0,0],[8.999999E+09,8.999999E+09,8.999999E+09,8.999999E+09,8.999999E+09,8.999999E+09]];
    LOCAL CONST Robtarget Tr_meulage_motif_1_152 := [[-47.378203125,19.385263671875,56.1948125],[0.325394831809823,-0.323189731818736,0.626217671016949,-0.630490308557156],[0,0,0,0],[8.999999E+09,8.999999E+09,8.999999E+09,8.999999E+09,8.999999E+09,8.999999E+09]];
    LOCAL CONST Robtarget Tr_meulage_motif_1_153 := [[-46.75214453125,20.35962109375,55.70727734375],[0.325394831809823,-0.323189731818736,0.626217671016949,-0.630490308557156],[0,0,0,0],[8.999999E+09,8.999999E+09,8.999999E+09,8.999999E+09,8.999999E+09,8.999999E+09]];
    LOCAL CONST Robtarget Tr_meulage_motif_1_154 := [[-46.29562109375,21.070720703125,55.4431796875],[0.325394831809823,-0.323189731818736,0.626217671016949,-0.630490308557156],[0,0,0,0],[8.999999E+09,8.999999E+09,8.999999E+09,8.999999E+09,8.999999E+09,8.999999E+09]];
    LOCAL CONST Robtarget Tr_meulage_motif_1_155 := [[-45.79237890625,21.855173828125,55.23870703125],[0.325394831809823,-0.323189731818736,0.626217671016949,-0.630490308557156],[0,0,0,0],[8.999999E+09,8.999999E+09,8.999999E+09,8.999999E+09,8.999999E+09,8.999999E+09]];
    LOCAL CONST Robtarget Tr_meulage_motif_1_156 := [[-45.26269140625,22.681548828125,55.13010546875],[0.325394831809823,-0.323189731818736,0.626217671016949,-0.630490308557156],[0,0,0,0],[8.999999E+09,8.999999E+09,8.999999E+09,8.999999E+09,8.999999E+09,8.999999E+09]];
    LOCAL CONST Robtarget Tr_meulage_motif_1_157 := [[-44.72706640625,23.51718359375,55.0195078125],[0.325394831809823,-0.323189731818736,0.626217671016949,-0.630490308557156],[0,0,0,0],[8.999999E+09,8.999999E+09,8.999999E+09,8.999999E+09,8.999999E+09,8.999999E+09]];
    LOCAL CONST Robtarget Tr_meulage_motif_1_158 := [[-44.18776171875,24.359294921875,55.0195],[0.325394831809823,-0.323189731818736,0.626217671016949,-0.630490308557156],[0,0,0,0],[8.999999E+09,8.999999E+09,8.999999E+09,8.999999E+09,8.999999E+09,8.999999E+09]];
    LOCAL CONST Robtarget Tr_meulage_motif_1_159 := [[-43.648453125,25.201404296875,55.01949609375],[0.325394831809823,-0.323189731818736,0.626217671016949,-0.630490308557156],[0,0,0,0],[8.999999E+09,8.999999E+09,8.999999E+09,8.999999E+09,8.999999E+09,8.999999E+09]];
    LOCAL CONST Robtarget Tr_meulage_motif_1_160 := [[-43.1091484375,26.043515625,55.01948828125],[0.325394831809823,-0.323189731818736,0.626217671016949,-0.630490308557156],[0,0,0,0],[8.999999E+09,8.999999E+09,8.999999E+09,8.999999E+09,8.999999E+09,8.999999E+09]];
    LOCAL CONST Robtarget Tr_meulage_motif_1_161 := [[-42.56984375,26.885625,55.019484375],[0.325394831809823,-0.323189731818736,0.626217671016949,-0.630490308557156],[0,0,0,0],[8.999999E+09,8.999999E+09,8.999999E+09,8.999999E+09,8.999999E+09,8.999999E+09]];
    LOCAL CONST Robtarget Tr_meulage_motif_1_162 := [[-42.0305390625,27.727736328125,55.0194765625],[0.325394831809823,-0.323189731818736,0.626217671016949,-0.630490308557156],[0,0,0,0],[8.999999E+09,8.999999E+09,8.999999E+09,8.999999E+09,8.999999E+09,8.999999E+09]];
    LOCAL CONST Robtarget Tr_meulage_motif_1_163 := [[-41.491234375,28.569845703125,55.01946875],[0.325394831809823,-0.323189731818736,0.626217671016949,-0.630490308557156],[0,0,0,0],[8.999999E+09,8.999999E+09,8.999999E+09,8.999999E+09,8.999999E+09,8.999999E+09]];
    LOCAL CONST Robtarget Tr_meulage_motif_1_164 := [[-40.9519296875,29.41195703125,55.01946484375],[0.325394831809823,-0.323189731818736,0.626217671016949,-0.630490308557156],[0,0,0,0],[8.999999E+09,8.999999E+09,8.999999E+09,8.999999E+09,8.999999E+09,8.999999E+09]];
    LOCAL CONST Robtarget Tr_meulage_motif_1_165 := [[-40.412625,30.254068359375,55.01945703125],[0.325394831809823,-0.323189731818736,0.626217671016949,-0.630490308557156],[0,0,0,0],[8.999999E+09,8.999999E+09,8.999999E+09,8.999999E+09,8.999999E+09,8.999999E+09]];
    LOCAL CONST Robtarget Tr_meulage_motif_1_166 := [[-39.8733203125,31.096177734375,55.01944921875],[0.325394831809823,-0.323189731818736,0.626217671016949,-0.630490308557156],[0,0,0,0],[8.999999E+09,8.999999E+09,8.999999E+09,8.999999E+09,8.999999E+09,8.999999E+09]];
    LOCAL CONST Robtarget Tr_meulage_motif_1_167 := [[-39.334015625,31.9382890625,55.0194453125],[0.325394831809823,-0.323189731818736,0.626217671016949,-0.630490308557156],[0,0,0,0],[8.999999E+09,8.999999E+09,8.999999E+09,8.999999E+09,8.999999E+09,8.999999E+09]];
    LOCAL CONST Robtarget Tr_meulage_motif_1_168 := [[-38.7947109375,32.7803984375,55.0194375],[0.325394831809823,-0.323189731818736,0.626217671016949,-0.630490308557156],[0,0,0,0],[8.999999E+09,8.999999E+09,8.999999E+09,8.999999E+09,8.999999E+09,8.999999E+09]];
    LOCAL CONST Robtarget Tr_meulage_motif_1_169 := [[-38.25540625,33.6225078125,55.01943359375],[0.325394831809823,-0.323189731818736,0.626217671016949,-0.630490308557156],[0,0,0,0],[8.999999E+09,8.999999E+09,8.999999E+09,8.999999E+09,8.999999E+09,8.999999E+09]];
    LOCAL CONST Robtarget Tr_meulage_motif_1_170 := [[-37.7161015625,34.46462109375,55.01942578125],[0.325394831809823,-0.323189731818736,0.626217671016949,-0.630490308557156],[0,0,0,0],[8.999999E+09,8.999999E+09,8.999999E+09,8.999999E+09,8.999999E+09,8.999999E+09]];
    LOCAL CONST Robtarget Tr_meulage_motif_1_171 := [[-37.17679296875,35.30673046875,55.01941796875],[0.325394831809823,-0.323189731818736,0.626217671016949,-0.630490308557156],[0,0,0,0],[8.999999E+09,8.999999E+09,8.999999E+09,8.999999E+09,8.999999E+09,8.999999E+09]];
    LOCAL CONST Robtarget Tr_meulage_motif_1_172 := [[-36.63748828125,36.14883984375,55.0194140625],[0.325394831809823,-0.323189731818736,0.626217671016949,-0.630490308557156],[0,0,0,0],[8.999999E+09,8.999999E+09,8.999999E+09,8.999999E+09,8.999999E+09,8.999999E+09]];
    LOCAL CONST Robtarget Tr_meulage_motif_1_173 := [[-36.09818359375,36.990953125,55.01940625],[0.325394831809823,-0.323189731818736,0.626217671016949,-0.630490308557156],[0,0,0,0],[8.999999E+09,8.999999E+09,8.999999E+09,8.999999E+09,8.999999E+09,8.999999E+09]];
    LOCAL CONST Robtarget Tr_meulage_motif_1_174 := [[-35.55887890625,37.8330625,55.01940234375],[0.325394831809823,-0.323189731818736,0.626217671016949,-0.630490308557156],[0,0,0,0],[8.999999E+09,8.999999E+09,8.999999E+09,8.999999E+09,8.999999E+09,8.999999E+09]];
    LOCAL CONST Robtarget Tr_meulage_motif_1_175 := [[-35.01957421875,38.675171875,55.01939453125],[0.325394831809823,-0.323189731818736,0.626217671016949,-0.630490308557156],[0,0,0,0],[8.999999E+09,8.999999E+09,8.999999E+09,8.999999E+09,8.999999E+09,8.999999E+09]];
    LOCAL CONST Robtarget Tr_meulage_motif_1_176 := [[-34.48026953125,39.51728515625,55.01938671875],[0.325394831809823,-0.323189731818736,0.626217671016949,-0.630490308557156],[0,0,0,0],[8.999999E+09,8.999999E+09,8.999999E+09,8.999999E+09,8.999999E+09,8.999999E+09]];
    LOCAL CONST Robtarget Tr_meulage_motif_1_177 := [[-33.94096484375,40.35939453125,55.0193828125],[0.325394831809823,-0.323189731818736,0.626217671016949,-0.630490308557156],[0,0,0,0],[8.999999E+09,8.999999E+09,8.999999E+09,8.999999E+09,8.999999E+09,8.999999E+09]];
    LOCAL CONST Robtarget Tr_meulage_motif_1_178 := [[-33.40166015625,41.20150390625,55.019375],[0.325394831809823,-0.323189731818736,0.626217671016949,-0.630490308557156],[0,0,0,0],[8.999999E+09,8.999999E+09,8.999999E+09,8.999999E+09,8.999999E+09,8.999999E+09]];
    LOCAL CONST Robtarget Tr_meulage_motif_1_179 := [[-32.86235546875,42.04361328125,55.0193671875],[0.325394831809823,-0.323189731818736,0.626217671016949,-0.630490308557156],[0,0,0,0],[8.999999E+09,8.999999E+09,8.999999E+09,8.999999E+09,8.999999E+09,8.999999E+09]];
    LOCAL CONST Robtarget Tr_meulage_motif_1_180 := [[-32.32305078125,42.8857265625,55.01936328125],[0.325394831809823,-0.323189731818736,0.626217671016949,-0.630490308557156],[0,0,0,0],[8.999999E+09,8.999999E+09,8.999999E+09,8.999999E+09,8.999999E+09,8.999999E+09]];
    LOCAL CONST Robtarget Tr_meulage_motif_1_181 := [[-31.783744140625,43.7278359375,55.01935546875],[0.325394831809823,-0.323189731818736,0.626217671016949,-0.630490308557156],[0,0,0,0],[8.999999E+09,8.999999E+09,8.999999E+09,8.999999E+09,8.999999E+09,8.999999E+09]];
    LOCAL CONST Robtarget Tr_meulage_motif_1_182 := [[-31.244439453125,44.5699453125,55.0193515625],[0.325394831809823,-0.323189731818736,0.626217671016949,-0.630490308557156],[0,0,0,0],[8.999999E+09,8.999999E+09,8.999999E+09,8.999999E+09,8.999999E+09,8.999999E+09]];
    LOCAL CONST Robtarget Tr_meulage_motif_1_183 := [[-30.705134765625,45.41205859375,55.01934375],[0.325394831809823,-0.323189731818736,0.626217671016949,-0.630490308557156],[0,0,0,0],[8.999999E+09,8.999999E+09,8.999999E+09,8.999999E+09,8.999999E+09,8.999999E+09]];
    LOCAL CONST Robtarget Tr_meulage_motif_1_184 := [[-30.165830078125,46.25416796875,55.0193359375],[0.325394831809823,-0.323189731818736,0.626217671016949,-0.630490308557156],[0,0,0,0],[8.999999E+09,8.999999E+09,8.999999E+09,8.999999E+09,8.999999E+09,8.999999E+09]];
    LOCAL CONST Robtarget Tr_meulage_motif_1_185 := [[-29.626525390625,47.09627734375,55.01933203125],[0.325394831809823,-0.323189731818736,0.626217671016949,-0.630490308557156],[0,0,0,0],[8.999999E+09,8.999999E+09,8.999999E+09,8.999999E+09,8.999999E+09,8.999999E+09]];
    LOCAL CONST Robtarget Tr_meulage_motif_1_186 := [[-29.087220703125,47.93838671875,55.01932421875],[0.325394831809823,-0.323189731818736,0.626217671016949,-0.630490308557156],[0,0,0,0],[8.999999E+09,8.999999E+09,8.999999E+09,8.999999E+09,8.999999E+09,8.999999E+09]];
    LOCAL CONST Robtarget Tr_meulage_motif_1_187 := [[-28.5479140625,48.7805,55.0193203125],[0.325394831809823,-0.323189731818736,0.626217671016949,-0.630490308557156],[0,0,0,0],[8.999999E+09,8.999999E+09,8.999999E+09,8.999999E+09,8.999999E+09,8.999999E+09]];
    LOCAL CONST Robtarget Tr_meulage_motif_1_188 := [[-28.0122890625,49.6161328125,54.90871875],[0.325394831809823,-0.323189731818736,0.626217671016949,-0.630490308557156],[0,0,0,0],[8.999999E+09,8.999999E+09,8.999999E+09,8.999999E+09,8.999999E+09,8.999999E+09]];
    LOCAL CONST Robtarget Tr_meulage_motif_1_189 := [[-27.501205078125,50.41278515625,54.69752734375],[0.325394831809823,-0.323189731818736,0.626217671016949,-0.630490308557156],[0,0,0,0],[8.999999E+09,8.999999E+09,8.999999E+09,8.999999E+09,8.999999E+09,8.999999E+09]];
    LOCAL CONST Robtarget Tr_meulage_motif_1_190 := [[-27.040515625,51.13034375,54.4256796875],[0.325394831809823,-0.323189731818736,0.626217671016949,-0.630490308557156],[0,0,0,0],[8.999999E+09,8.999999E+09,8.999999E+09,8.999999E+09,8.999999E+09,8.999999E+09]];
    LOCAL CONST Robtarget Tr_meulage_motif_1_191 := [[-26.655888671875,51.72891796875,54.12153515625],[0.325394831809823,-0.323189731818736,0.626217671016949,-0.630490308557156],[0,0,0,0],[8.999999E+09,8.999999E+09,8.999999E+09,8.999999E+09,8.999999E+09,8.999999E+09]];
    LOCAL CONST Robtarget Tr_meulage_motif_1_192 := [[-26.0960078125,52.59878125,53.45900390625],[0.325394831809823,-0.323189731818736,0.626217671016949,-0.630490308557156],[0,0,0,0],[8.999999E+09,8.999999E+09,8.999999E+09,8.999999E+09,8.999999E+09,8.999999E+09]];
    LOCAL CONST Robtarget Tr_meulage_motif_1_193 := [[-25.60688671875,53.35657421875,52.55705078125],[0.325394831809823,-0.323189731818736,0.626217671016949,-0.630490308557156],[0,0,0,0],[8.999999E+09,8.999999E+09,8.999999E+09,8.999999E+09,8.999999E+09,8.999999E+09]];
    LOCAL CONST Robtarget Tr_meulage_motif_1_194 := [[-25.3152421875,53.8050625,51.5110390625],[0.325394831809823,-0.323189731818736,0.626217671016949,-0.630490308557156],[0,0,0,0],[8.999999E+09,8.999999E+09,8.999999E+09,8.999999E+09,8.999999E+09,8.999999E+09]];
    LOCAL CONST Robtarget Tr_meulage_motif_1_195 := [[-25.213509765625,53.95933203125,50.8178046875],[0.325394831809823,-0.323189731818736,0.626217671016949,-0.630490308557156],[0,0,0,0],[8.999999E+09,8.999999E+09,8.999999E+09,8.999999E+09,8.999999E+09,8.999999E+09]];
    LOCAL CONST Robtarget Tr_meulage_motif_1_196 := [[-25.176771484375,54.01161328125,50.0478125],[0.325394831809823,-0.323189731818736,0.626217671016949,-0.630490308557156],[0,0,0,0],[8.999999E+09,8.999999E+09,8.999999E+09,8.999999E+09,8.999999E+09,8.999999E+09]];
    LOCAL CONST Robtarget Tr_meulage_motif_1_197 := [[-25.210564453125,53.95376171875,49.27795703125],[0.325394831809823,-0.323189731818736,0.626217671016949,-0.630490308557156],[0,0,0,0],[8.999999E+09,8.999999E+09,8.999999E+09,8.999999E+09,8.999999E+09,8.999999E+09]];
    LOCAL CONST Robtarget Tr_meulage_motif_1_198 := [[-25.433533203125,53.59828125,48.16971484375],[0.325394831809823,-0.323189731818736,0.626217671016949,-0.630490308557156],[0,0,0,0],[8.999999E+09,8.999999E+09,8.999999E+09,8.999999E+09,8.999999E+09,8.999999E+09]];
    LOCAL CONST Robtarget Tr_meulage_motif_1_199 := [[-25.65521875,53.2482578125,47.58403515625],[0.325394831809823,-0.323189731818736,0.626217671016949,-0.630490308557156],[0,0,0,0],[8.999999E+09,8.999999E+09,8.999999E+09,8.999999E+09,8.999999E+09,8.999999E+09]];
    LOCAL CONST Robtarget Tr_meulage_motif_1_200 := [[-26.1309921875,52.4994921875,46.696890625],[0.325394831809823,-0.323189731818736,0.626217671016949,-0.630490308557156],[0,0,0,0],[8.999999E+09,8.999999E+09,8.999999E+09,8.999999E+09,8.999999E+09,8.999999E+09]];
    LOCAL CONST Robtarget Tr_meulage_motif_1_201 := [[-26.445615234375,52.00548046875,46.2826171875],[0.325394831809823,-0.323189731818736,0.626217671016949,-0.630490308557156],[0,0,0,0],[8.999999E+09,8.999999E+09,8.999999E+09,8.999999E+09,8.999999E+09,8.999999E+09]];
    LOCAL CONST Robtarget Tr_meulage_motif_1_202 := [[-27.046876953125,51.06303125,45.7385],[0.325394831809823,-0.323189731818736,0.626217671016949,-0.630490308557156],[0,0,0,0],[8.999999E+09,8.999999E+09,8.999999E+09,8.999999E+09,8.999999E+09,8.999999E+09]];
    LOCAL CONST Robtarget Tr_meulage_motif_1_203 := [[-27.49123828125,50.36721875,45.4430078125],[0.325394831809823,-0.323189731818736,0.626217671016949,-0.630490308557156],[0,0,0,0],[8.999999E+09,8.999999E+09,8.999999E+09,8.999999E+09,8.999999E+09,8.999999E+09]];
    LOCAL CONST Robtarget Tr_meulage_motif_1_204 := [[-27.9932578125,49.5819765625,45.23853125],[0.325394831809823,-0.323189731818736,0.626217671016949,-0.630490308557156],[0,0,0,0],[8.999999E+09,8.999999E+09,8.999999E+09,8.999999E+09,8.999999E+09,8.999999E+09]];
    LOCAL CONST Robtarget Tr_meulage_motif_1_205 := [[-28.522294921875,48.75518359375,45.1299921875],[0.325394831809823,-0.323189731818736,0.626217671016949,-0.630490308557156],[0,0,0,0],[8.999999E+09,8.999999E+09,8.999999E+09,8.999999E+09,8.999999E+09,8.999999E+09]];
    LOCAL CONST Robtarget Tr_meulage_motif_1_206 := [[-29.0572578125,47.919125,45.01938671875],[0.325394831809823,-0.323189731818736,0.626217671016949,-0.630490308557156],[0,0,0,0],[8.999999E+09,8.999999E+09,8.999999E+09,8.999999E+09,8.999999E+09,8.999999E+09]];
    LOCAL CONST Robtarget Tr_meulage_motif_1_207 := [[-29.5965625,47.077015625,45.01939453125],[0.325394831809823,-0.323189731818736,0.626217671016949,-0.630490308557156],[0,0,0,0],[8.999999E+09,8.999999E+09,8.999999E+09,8.999999E+09,8.999999E+09,8.999999E+09]];
    LOCAL CONST Robtarget Tr_meulage_motif_1_208 := [[-30.1358671875,46.23490234375,45.01940234375],[0.325394831809823,-0.323189731818736,0.626217671016949,-0.630490308557156],[0,0,0,0],[8.999999E+09,8.999999E+09,8.999999E+09,8.999999E+09,8.999999E+09,8.999999E+09]];
    LOCAL CONST Robtarget Tr_meulage_motif_1_209 := [[-30.675171875,45.39279296875,45.01940625],[0.325394831809823,-0.323189731818736,0.626217671016949,-0.630490308557156],[0,0,0,0],[8.999999E+09,8.999999E+09,8.999999E+09,8.999999E+09,8.999999E+09,8.999999E+09]];
    LOCAL CONST Robtarget Tr_meulage_motif_1_210 := [[-31.2144765625,44.55068359375,45.0194140625],[0.325394831809823,-0.323189731818736,0.626217671016949,-0.630490308557156],[0,0,0,0],[8.999999E+09,8.999999E+09,8.999999E+09,8.999999E+09,8.999999E+09,8.999999E+09]];
    LOCAL CONST Robtarget Tr_meulage_motif_1_211 := [[-31.753783203125,43.70857421875,45.01941796875],[0.325394831809823,-0.323189731818736,0.626217671016949,-0.630490308557156],[0,0,0,0],[8.999999E+09,8.999999E+09,8.999999E+09,8.999999E+09,8.999999E+09,8.999999E+09]];
    LOCAL CONST Robtarget Tr_meulage_motif_1_212 := [[-32.293087890625,42.8664609375,45.01942578125],[0.325394831809823,-0.323189731818736,0.626217671016949,-0.630490308557156],[0,0,0,0],[8.999999E+09,8.999999E+09,8.999999E+09,8.999999E+09,8.999999E+09,8.999999E+09]];
    LOCAL CONST Robtarget Tr_meulage_motif_1_213 := [[-32.832390625,42.0243515625,45.01943359375],[0.325394831809823,-0.323189731818736,0.626217671016949,-0.630490308557156],[0,0,0,0],[8.999999E+09,8.999999E+09,8.999999E+09,8.999999E+09,8.999999E+09,8.999999E+09]];
    LOCAL CONST Robtarget Tr_meulage_motif_1_214 := [[-33.37169921875,41.1822421875,45.0194375],[0.325394831809823,-0.323189731818736,0.626217671016949,-0.630490308557156],[0,0,0,0],[8.999999E+09,8.999999E+09,8.999999E+09,8.999999E+09,8.999999E+09,8.999999E+09]];
    LOCAL CONST Robtarget Tr_meulage_motif_1_215 := [[-33.91100390625,40.34012890625,45.0194453125],[0.325394831809823,-0.323189731818736,0.626217671016949,-0.630490308557156],[0,0,0,0],[8.999999E+09,8.999999E+09,8.999999E+09,8.999999E+09,8.999999E+09,8.999999E+09]];
    LOCAL CONST Robtarget Tr_meulage_motif_1_216 := [[-34.45030859375,39.49801953125,45.019453125],[0.325394831809823,-0.323189731818736,0.626217671016949,-0.630490308557156],[0,0,0,0],[8.999999E+09,8.999999E+09,8.999999E+09,8.999999E+09,8.999999E+09,8.999999E+09]];
    LOCAL CONST Robtarget Tr_meulage_motif_1_217 := [[-34.98961328125,38.65591015625,45.01945703125],[0.325394831809823,-0.323189731818736,0.626217671016949,-0.630490308557156],[0,0,0,0],[8.999999E+09,8.999999E+09,8.999999E+09,8.999999E+09,8.999999E+09,8.999999E+09]];
    LOCAL CONST Robtarget Tr_meulage_motif_1_218 := [[-35.52891796875,37.813796875,45.01946484375],[0.325394831809823,-0.323189731818736,0.626217671016949,-0.630490308557156],[0,0,0,0],[8.999999E+09,8.999999E+09,8.999999E+09,8.999999E+09,8.999999E+09,8.999999E+09]];
    LOCAL CONST Robtarget Tr_meulage_motif_1_219 := [[-36.06822265625,36.9716875,45.01946875],[0.325394831809823,-0.323189731818736,0.626217671016949,-0.630490308557156],[0,0,0,0],[8.999999E+09,8.999999E+09,8.999999E+09,8.999999E+09,8.999999E+09,8.999999E+09]];
    LOCAL CONST Robtarget Tr_meulage_motif_1_220 := [[-36.60752734375,36.129578125,45.0194765625],[0.325394831809823,-0.323189731818736,0.626217671016949,-0.630490308557156],[0,0,0,0],[8.999999E+09,8.999999E+09,8.999999E+09,8.999999E+09,8.999999E+09,8.999999E+09]];
    LOCAL CONST Robtarget Tr_meulage_motif_1_221 := [[-37.14683203125,35.28746875,45.019484375],[0.325394831809823,-0.323189731818736,0.626217671016949,-0.630490308557156],[0,0,0,0],[8.999999E+09,8.999999E+09,8.999999E+09,8.999999E+09,8.999999E+09,8.999999E+09]];
    LOCAL CONST Robtarget Tr_meulage_motif_1_222 := [[-37.68613671875,34.44535546875,45.01948828125],[0.325394831809823,-0.323189731818736,0.626217671016949,-0.630490308557156],[0,0,0,0],[8.999999E+09,8.999999E+09,8.999999E+09,8.999999E+09,8.999999E+09,8.999999E+09]];
    LOCAL CONST Robtarget Tr_meulage_motif_1_223 := [[-38.22544140625,33.60324609375,45.01949609375],[0.325394831809823,-0.323189731818736,0.626217671016949,-0.630490308557156],[0,0,0,0],[8.999999E+09,8.999999E+09,8.999999E+09,8.999999E+09,8.999999E+09,8.999999E+09]];
    LOCAL CONST Robtarget Tr_meulage_motif_1_224 := [[-38.76474609375,32.761134765625,45.0195],[0.325394831809823,-0.323189731818736,0.626217671016949,-0.630490308557156],[0,0,0,0],[8.999999E+09,8.999999E+09,8.999999E+09,8.999999E+09,8.999999E+09,8.999999E+09]];
    LOCAL CONST Robtarget Tr_meulage_motif_1_225 := [[-39.30405078125,31.919025390625,45.0195078125],[0.325394831809823,-0.323189731818736,0.626217671016949,-0.630490308557156],[0,0,0,0],[8.999999E+09,8.999999E+09,8.999999E+09,8.999999E+09,8.999999E+09,8.999999E+09]];
    LOCAL CONST Robtarget Tr_meulage_motif_1_226 := [[-39.84335546875,31.0769140625,45.019515625],[0.325394831809823,-0.323189731818736,0.626217671016949,-0.630490308557156],[0,0,0,0],[8.999999E+09,8.999999E+09,8.999999E+09,8.999999E+09,8.999999E+09,8.999999E+09]];
    LOCAL CONST Robtarget Tr_meulage_motif_1_227 := [[-40.3826640625,30.2348046875,45.01951953125],[0.325394831809823,-0.323189731818736,0.626217671016949,-0.630490308557156],[0,0,0,0],[8.999999E+09,8.999999E+09,8.999999E+09,8.999999E+09,8.999999E+09,8.999999E+09]];
    LOCAL CONST Robtarget Tr_meulage_motif_1_228 := [[-40.92196875,29.392693359375,45.01952734375],[0.325394831809823,-0.323189731818736,0.626217671016949,-0.630490308557156],[0,0,0,0],[8.999999E+09,8.999999E+09,8.999999E+09,8.999999E+09,8.999999E+09,8.999999E+09]];
    LOCAL CONST Robtarget Tr_meulage_motif_1_229 := [[-41.4612734375,28.550583984375,45.01953515625],[0.325394831809823,-0.323189731818736,0.626217671016949,-0.630490308557156],[0,0,0,0],[8.999999E+09,8.999999E+09,8.999999E+09,8.999999E+09,8.999999E+09,8.999999E+09]];
    LOCAL CONST Robtarget Tr_meulage_motif_1_230 := [[-42.000578125,27.70847265625,45.0195390625],[0.325394831809823,-0.323189731818736,0.626217671016949,-0.630490308557156],[0,0,0,0],[8.999999E+09,8.999999E+09,8.999999E+09,8.999999E+09,8.999999E+09,8.999999E+09]];
    LOCAL CONST Robtarget Tr_meulage_motif_1_231 := [[-42.5398828125,26.866361328125,45.019546875],[0.325394831809823,-0.323189731818736,0.626217671016949,-0.630490308557156],[0,0,0,0],[8.999999E+09,8.999999E+09,8.999999E+09,8.999999E+09,8.999999E+09,8.999999E+09]];
    LOCAL CONST Robtarget Tr_meulage_motif_1_232 := [[-43.0791875,26.024251953125,45.01955078125],[0.325394831809823,-0.323189731818736,0.626217671016949,-0.630490308557156],[0,0,0,0],[8.999999E+09,8.999999E+09,8.999999E+09,8.999999E+09,8.999999E+09,8.999999E+09]];
    LOCAL CONST Robtarget Tr_meulage_motif_1_233 := [[-43.6184921875,25.182140625,45.01955859375],[0.325394831809823,-0.323189731818736,0.626217671016949,-0.630490308557156],[0,0,0,0],[8.999999E+09,8.999999E+09,8.999999E+09,8.999999E+09,8.999999E+09,8.999999E+09]];
    LOCAL CONST Robtarget Tr_meulage_motif_1_234 := [[-44.157796875,24.34003125,45.01956640625],[0.325394831809823,-0.323189731818736,0.626217671016949,-0.630490308557156],[0,0,0,0],[8.999999E+09,8.999999E+09,8.999999E+09,8.999999E+09,8.999999E+09,8.999999E+09]];
    LOCAL CONST Robtarget Tr_meulage_motif_1_235 := [[-44.6971015625,23.497919921875,45.0195703125],[0.325394831809823,-0.323189731818736,0.626217671016949,-0.630490308557156],[0,0,0,0],[8.999999E+09,8.999999E+09,8.999999E+09,8.999999E+09,8.999999E+09,8.999999E+09]];
    LOCAL CONST Robtarget Tr_meulage_motif_1_236 := [[-45.23640625,22.65580859375,45.019578125],[0.325394831809823,-0.323189731818736,0.626217671016949,-0.630490308557156],[0,0,0,0],[8.999999E+09,8.999999E+09,8.999999E+09,8.999999E+09,8.999999E+09,8.999999E+09]];
    LOCAL CONST Robtarget Tr_meulage_motif_1_237 := [[-45.77137109375,21.81975,44.9089765625],[0.325394831809823,-0.323189731818736,0.626217671016949,-0.630490308557156],[0,0,0,0],[8.999999E+09,8.999999E+09,8.999999E+09,8.999999E+09,8.999999E+09,8.999999E+09]];
    LOCAL CONST Robtarget Tr_meulage_motif_1_238 := [[-46.2811875,21.02228515625,44.69779296875],[0.325394831809823,-0.323189731818736,0.626217671016949,-0.630490308557156],[0,0,0,0],[8.999999E+09,8.999999E+09,8.999999E+09,8.999999E+09,8.999999E+09,8.999999E+09]];
    LOCAL CONST Robtarget Tr_meulage_motif_1_239 := [[-46.74025,20.303677734375,44.42597265625],[0.325394831809823,-0.323189731818736,0.626217671016949,-0.630490308557156],[0,0,0,0],[8.999999E+09,8.999999E+09,8.999999E+09,8.999999E+09,8.999999E+09,8.999999E+09]];
    LOCAL CONST Robtarget Tr_meulage_motif_1_240 := [[-47.1230546875,19.7039296875,44.12183984375],[0.325394831809823,-0.323189731818736,0.626217671016949,-0.630490308557156],[0,0,0,0],[8.999999E+09,8.999999E+09,8.999999E+09,8.999999E+09,8.999999E+09,8.999999E+09]];
    LOCAL CONST Robtarget Tr_meulage_motif_1_241 := [[-47.67896484375,18.831517578125,43.4593203125],[0.325394831809823,-0.323189731818736,0.626217671016949,-0.630490308557156],[0,0,0,0],[8.999999E+09,8.999999E+09,8.999999E+09,8.999999E+09,8.999999E+09,8.999999E+09]];
    LOCAL CONST Robtarget Tr_meulage_motif_1_242 := [[-48.11453515625,18.14517578125,42.51955078125],[0.325394831809823,-0.323189731818736,0.626217671016949,-0.630490308557156],[0,0,0,0],[8.999999E+09,8.999999E+09,8.999999E+09,8.999999E+09,8.999999E+09,8.999999E+09]];
    LOCAL CONST Robtarget Tr_meulage_motif_1_243 := [[-48.30162109375,17.84646484375,41.52319921875],[0.325394831809823,-0.323189731818736,0.626217671016949,-0.630490308557156],[0,0,0,0],[8.999999E+09,8.999999E+09,8.999999E+09,8.999999E+09,8.999999E+09,8.999999E+09]];
    LOCAL CONST Robtarget Tr_meulage_motif_1_244 := [[-48.28395703125,17.870365234375,40.96565625],[0.325394831809823,-0.323189731818736,0.626217671016949,-0.630490308557156],[0,0,0,0],[8.999999E+09,8.999999E+09,8.999999E+09,8.999999E+09,8.999999E+09,8.999999E+09]];
    LOCAL CONST Robtarget Tr_meulage_motif_1_245 := [[-48.28503125,17.865927734375,40.54775],[0.325394831809823,-0.323189731818736,0.626217671016949,-0.630490308557156],[0,0,0,0],[8.999999E+09,8.999999E+09,8.999999E+09,8.999999E+09,8.999999E+09,8.999999E+09]];
    LOCAL CONST Robtarget Tr_meulage_motif_1_246 := [[-48.0868125,18.169037109375,39.57842578125],[0.325394831809823,-0.323189731818736,0.626217671016949,-0.630490308557156],[0,0,0,0],[8.999999E+09,8.999999E+09,8.999999E+09,8.999999E+09,8.999999E+09,8.999999E+09]];
    LOCAL CONST Robtarget Tr_meulage_motif_1_247 := [[-47.6407890625,18.859431640625,38.66073828125],[0.325394831809823,-0.323189731818736,0.626217671016949,-0.630490308557156],[0,0,0,0],[8.999999E+09,8.999999E+09,8.999999E+09,8.999999E+09,8.999999E+09,8.999999E+09]];
    LOCAL CONST Robtarget Tr_meulage_motif_1_248 := [[-47.3093828125,19.374119140625,38.23784765625],[0.325394831809823,-0.323189731818736,0.626217671016949,-0.630490308557156],[0,0,0,0],[8.999999E+09,8.999999E+09,8.999999E+09,8.999999E+09,8.999999E+09,8.999999E+09]];
    LOCAL CONST Robtarget Tr_meulage_motif_1_249 := [[-46.6982109375,20.3249453125,37.707390625],[0.325394831809823,-0.323189731818736,0.626217671016949,-0.630490308557156],[0,0,0,0],[8.999999E+09,8.999999E+09,8.999999E+09,8.999999E+09,8.999999E+09,8.999999E+09]];
    LOCAL CONST Robtarget Tr_meulage_motif_1_250 := [[-46.2416875,21.036046875,37.44327734375],[0.325394831809823,-0.323189731818736,0.626217671016949,-0.630490308557156],[0,0,0,0],[8.999999E+09,8.999999E+09,8.999999E+09,8.999999E+09,8.999999E+09,8.999999E+09]];
    LOCAL CONST Robtarget Tr_meulage_motif_1_251 := [[-45.7384453125,21.8205,37.2387890625],[0.325394831809823,-0.323189731818736,0.626217671016949,-0.630490308557156],[0,0,0,0],[8.999999E+09,8.999999E+09,8.999999E+09,8.999999E+09,8.999999E+09,8.999999E+09]];
    LOCAL CONST Robtarget Tr_meulage_motif_1_252 := [[-45.2087578125,22.646875,37.13023828125],[0.325394831809823,-0.323189731818736,0.626217671016949,-0.630490308557156],[0,0,0,0],[8.999999E+09,8.999999E+09,8.999999E+09,8.999999E+09,8.999999E+09,8.999999E+09]];
    LOCAL CONST Robtarget Tr_meulage_motif_1_253 := [[-44.6731328125,23.482509765625,37.01962109375],[0.325394831809823,-0.323189731818736,0.626217671016949,-0.630490308557156],[0,0,0,0],[8.999999E+09,8.999999E+09,8.999999E+09,8.999999E+09,8.999999E+09,8.999999E+09]];
    LOCAL CONST Robtarget Tr_meulage_motif_1_254 := [[-44.133828125,24.324619140625,37.0196171875],[0.325394831809823,-0.323189731818736,0.626217671016949,-0.630490308557156],[0,0,0,0],[8.999999E+09,8.999999E+09,8.999999E+09,8.999999E+09,8.999999E+09,8.999999E+09]];
    LOCAL CONST Robtarget Tr_meulage_motif_1_255 := [[-43.5945234375,25.16673046875,37.019609375],[0.325394831809823,-0.323189731818736,0.626217671016949,-0.630490308557156],[0,0,0,0],[8.999999E+09,8.999999E+09,8.999999E+09,8.999999E+09,8.999999E+09,8.999999E+09]];
    LOCAL CONST Robtarget Tr_meulage_motif_1_256 := [[-43.05521875,26.00883984375,37.0196015625],[0.325394831809823,-0.323189731818736,0.626217671016949,-0.630490308557156],[0,0,0,0],[8.999999E+09,8.999999E+09,8.999999E+09,8.999999E+09,8.999999E+09,8.999999E+09]];
    LOCAL CONST Robtarget Tr_meulage_motif_1_257 := [[-42.5159140625,26.850951171875,37.01959765625],[0.325394831809823,-0.323189731818736,0.626217671016949,-0.630490308557156],[0,0,0,0],[8.999999E+09,8.999999E+09,8.999999E+09,8.999999E+09,8.999999E+09,8.999999E+09]];
    LOCAL CONST Robtarget Tr_meulage_motif_1_258 := [[-41.97660546875,27.6930625,37.01958984375],[0.325394831809823,-0.323189731818736,0.626217671016949,-0.630490308557156],[0,0,0,0],[8.999999E+09,8.999999E+09,8.999999E+09,8.999999E+09,8.999999E+09,8.999999E+09]];
    LOCAL CONST Robtarget Tr_meulage_motif_1_259 := [[-41.43730078125,28.535171875,37.0195859375],[0.325394831809823,-0.323189731818736,0.626217671016949,-0.630490308557156],[0,0,0,0],[8.999999E+09,8.999999E+09,8.999999E+09,8.999999E+09,8.999999E+09,8.999999E+09]];
    LOCAL CONST Robtarget Tr_meulage_motif_1_260 := [[-40.89799609375,29.377283203125,37.019578125],[0.325394831809823,-0.323189731818736,0.626217671016949,-0.630490308557156],[0,0,0,0],[8.999999E+09,8.999999E+09,8.999999E+09,8.999999E+09,8.999999E+09,8.999999E+09]];
    LOCAL CONST Robtarget Tr_meulage_motif_1_261 := [[-40.35869140625,30.219392578125,37.0195703125],[0.325394831809823,-0.323189731818736,0.626217671016949,-0.630490308557156],[0,0,0,0],[8.999999E+09,8.999999E+09,8.999999E+09,8.999999E+09,8.999999E+09,8.999999E+09]];
    LOCAL CONST Robtarget Tr_meulage_motif_1_262 := [[-39.81938671875,31.06150390625,37.01956640625],[0.325394831809823,-0.323189731818736,0.626217671016949,-0.630490308557156],[0,0,0,0],[8.999999E+09,8.999999E+09,8.999999E+09,8.999999E+09,8.999999E+09,8.999999E+09]];
    LOCAL CONST Robtarget Tr_meulage_motif_1_263 := [[-39.28008203125,31.903615234375,37.01955859375],[0.325394831809823,-0.323189731818736,0.626217671016949,-0.630490308557156],[0,0,0,0],[8.999999E+09,8.999999E+09,8.999999E+09,8.999999E+09,8.999999E+09,8.999999E+09]];
    LOCAL CONST Robtarget Tr_meulage_motif_1_264 := [[-38.74077734375,32.745724609375,37.01955078125],[0.325394831809823,-0.323189731818736,0.626217671016949,-0.630490308557156],[0,0,0,0],[8.999999E+09,8.999999E+09,8.999999E+09,8.999999E+09,8.999999E+09,8.999999E+09]];
    LOCAL CONST Robtarget Tr_meulage_motif_1_265 := [[-38.20147265625,33.5878359375,37.019546875],[0.325394831809823,-0.323189731818736,0.626217671016949,-0.630490308557156],[0,0,0,0],[8.999999E+09,8.999999E+09,8.999999E+09,8.999999E+09,8.999999E+09,8.999999E+09]];
    LOCAL CONST Robtarget Tr_meulage_motif_1_266 := [[-37.66216796875,34.4299453125,37.0195390625],[0.325394831809823,-0.323189731818736,0.626217671016949,-0.630490308557156],[0,0,0,0],[8.999999E+09,8.999999E+09,8.999999E+09,8.999999E+09,8.999999E+09,8.999999E+09]];
    LOCAL CONST Robtarget Tr_meulage_motif_1_267 := [[-37.12286328125,35.2720546875,37.01953515625],[0.325394831809823,-0.323189731818736,0.626217671016949,-0.630490308557156],[0,0,0,0],[8.999999E+09,8.999999E+09,8.999999E+09,8.999999E+09,8.999999E+09,8.999999E+09]];
    LOCAL CONST Robtarget Tr_meulage_motif_1_268 := [[-36.58355859375,36.11416796875,37.01952734375],[0.325394831809823,-0.323189731818736,0.626217671016949,-0.630490308557156],[0,0,0,0],[8.999999E+09,8.999999E+09,8.999999E+09,8.999999E+09,8.999999E+09,8.999999E+09]];
    LOCAL CONST Robtarget Tr_meulage_motif_1_269 := [[-36.04425390625,36.95627734375,37.01951953125],[0.325394831809823,-0.323189731818736,0.626217671016949,-0.630490308557156],[0,0,0,0],[8.999999E+09,8.999999E+09,8.999999E+09,8.999999E+09,8.999999E+09,8.999999E+09]];
    LOCAL CONST Robtarget Tr_meulage_motif_1_270 := [[-35.5049453125,37.79838671875,37.019515625],[0.325394831809823,-0.323189731818736,0.626217671016949,-0.630490308557156],[0,0,0,0],[8.999999E+09,8.999999E+09,8.999999E+09,8.999999E+09,8.999999E+09,8.999999E+09]];
    LOCAL CONST Robtarget Tr_meulage_motif_1_271 := [[-34.965640625,38.6405,37.0195078125],[0.325394831809823,-0.323189731818736,0.626217671016949,-0.630490308557156],[0,0,0,0],[8.999999E+09,8.999999E+09,8.999999E+09,8.999999E+09,8.999999E+09,8.999999E+09]];
    LOCAL CONST Robtarget Tr_meulage_motif_1_272 := [[-34.4263359375,39.482609375,37.01950390625],[0.325394831809823,-0.323189731818736,0.626217671016949,-0.630490308557156],[0,0,0,0],[8.999999E+09,8.999999E+09,8.999999E+09,8.999999E+09,8.999999E+09,8.999999E+09]];
    LOCAL CONST Robtarget Tr_meulage_motif_1_273 := [[-33.88703125,40.32471875,37.01949609375],[0.325394831809823,-0.323189731818736,0.626217671016949,-0.630490308557156],[0,0,0,0],[8.999999E+09,8.999999E+09,8.999999E+09,8.999999E+09,8.999999E+09,8.999999E+09]];
    LOCAL CONST Robtarget Tr_meulage_motif_1_274 := [[-33.3477265625,41.166828125,37.01948828125],[0.325394831809823,-0.323189731818736,0.626217671016949,-0.630490308557156],[0,0,0,0],[8.999999E+09,8.999999E+09,8.999999E+09,8.999999E+09,8.999999E+09,8.999999E+09]];
    LOCAL CONST Robtarget Tr_meulage_motif_1_275 := [[-32.808421875,42.00894140625,37.019484375],[0.325394831809823,-0.323189731818736,0.626217671016949,-0.630490308557156],[0,0,0,0],[8.999999E+09,8.999999E+09,8.999999E+09,8.999999E+09,8.999999E+09,8.999999E+09]];
    LOCAL CONST Robtarget Tr_meulage_motif_1_276 := [[-32.2691171875,42.85105078125,37.0194765625],[0.325394831809823,-0.323189731818736,0.626217671016949,-0.630490308557156],[0,0,0,0],[8.999999E+09,8.999999E+09,8.999999E+09,8.999999E+09,8.999999E+09,8.999999E+09]];
    LOCAL CONST Robtarget Tr_meulage_motif_1_277 := [[-31.7298125,43.69316015625,37.01946875],[0.325394831809823,-0.323189731818736,0.626217671016949,-0.630490308557156],[0,0,0,0],[8.999999E+09,8.999999E+09,8.999999E+09,8.999999E+09,8.999999E+09,8.999999E+09]];
    LOCAL CONST Robtarget Tr_meulage_motif_1_278 := [[-31.1905078125,44.5352734375,37.01946484375],[0.325394831809823,-0.323189731818736,0.626217671016949,-0.630490308557156],[0,0,0,0],[8.999999E+09,8.999999E+09,8.999999E+09,8.999999E+09,8.999999E+09,8.999999E+09]];
    LOCAL CONST Robtarget Tr_meulage_motif_1_279 := [[-30.651203125,45.3773828125,37.01945703125],[0.325394831809823,-0.323189731818736,0.626217671016949,-0.630490308557156],[0,0,0,0],[8.999999E+09,8.999999E+09,8.999999E+09,8.999999E+09,8.999999E+09,8.999999E+09]];
    LOCAL CONST Robtarget Tr_meulage_motif_1_280 := [[-30.111896484375,46.2194921875,37.019453125],[0.325394831809823,-0.323189731818736,0.626217671016949,-0.630490308557156],[0,0,0,0],[8.999999E+09,8.999999E+09,8.999999E+09,8.999999E+09,8.999999E+09,8.999999E+09]];
    LOCAL CONST Robtarget Tr_meulage_motif_1_281 := [[-29.572591796875,47.06160546875,37.0194453125],[0.325394831809823,-0.323189731818736,0.626217671016949,-0.630490308557156],[0,0,0,0],[8.999999E+09,8.999999E+09,8.999999E+09,8.999999E+09,8.999999E+09,8.999999E+09]];
    LOCAL CONST Robtarget Tr_meulage_motif_1_282 := [[-29.033287109375,47.90371484375,37.0194375],[0.325394831809823,-0.323189731818736,0.626217671016949,-0.630490308557156],[0,0,0,0],[8.999999E+09,8.999999E+09,8.999999E+09,8.999999E+09,8.999999E+09,8.999999E+09]];
    LOCAL CONST Robtarget Tr_meulage_motif_1_283 := [[-28.493982421875,48.74582421875,37.01943359375],[0.325394831809823,-0.323189731818736,0.626217671016949,-0.630490308557156],[0,0,0,0],[8.999999E+09,8.999999E+09,8.999999E+09,8.999999E+09,8.999999E+09,8.999999E+09]];
    LOCAL CONST Robtarget Tr_meulage_motif_1_284 := [[-27.954677734375,49.58793359375,37.01942578125],[0.325394831809823,-0.323189731818736,0.626217671016949,-0.630490308557156],[0,0,0,0],[8.999999E+09,8.999999E+09,8.999999E+09,8.999999E+09,8.999999E+09,8.999999E+09]];
    LOCAL CONST Robtarget Tr_meulage_motif_1_285 := [[-27.415373046875,50.430046875,37.019421875],[0.325394831809823,-0.323189731818736,0.626217671016949,-0.630490308557156],[0,0,0,0],[8.999999E+09,8.999999E+09,8.999999E+09,8.999999E+09,8.999999E+09,8.999999E+09]];
    LOCAL CONST Robtarget Tr_meulage_motif_1_286 := [[-26.87606640625,51.27215625,37.0194140625],[0.325394831809823,-0.323189731818736,0.626217671016949,-0.630490308557156],[0,0,0,0],[8.999999E+09,8.999999E+09,8.999999E+09,8.999999E+09,8.999999E+09,8.999999E+09]];
    LOCAL CONST Robtarget Tr_meulage_motif_1_287 := [[-26.33676171875,52.114265625,37.01940625],[0.325394831809823,-0.323189731818736,0.626217671016949,-0.630490308557156],[0,0,0,0],[8.999999E+09,8.999999E+09,8.999999E+09,8.999999E+09,8.999999E+09,8.999999E+09]];
    LOCAL CONST Robtarget Tr_meulage_motif_1_288 := [[-25.79745703125,52.95637890625,37.01940234375],[0.325394831809823,-0.323189731818736,0.626217671016949,-0.630490308557156],[0,0,0,0],[8.999999E+09,8.999999E+09,8.999999E+09,8.999999E+09,8.999999E+09,8.999999E+09]];
    LOCAL CONST Robtarget Tr_meulage_motif_1_289 := [[-25.25815234375,53.79848828125,37.01939453125],[0.325394831809823,-0.323189731818736,0.626217671016949,-0.630490308557156],[0,0,0,0],[8.999999E+09,8.999999E+09,8.999999E+09,8.999999E+09,8.999999E+09,8.999999E+09]];
    LOCAL CONST Robtarget Tr_meulage_motif_1_290 := [[-24.71884765625,54.64059765625,37.01938671875],[0.325394831809823,-0.323189731818736,0.626217671016949,-0.630490308557156],[0,0,0,0],[8.999999E+09,8.999999E+09,8.999999E+09,8.999999E+09,8.999999E+09,8.999999E+09]];
    LOCAL CONST Robtarget Tr_meulage_motif_1_291 := [[-24.17954296875,55.48270703125,37.0193828125],[0.325394831809823,-0.323189731818736,0.626217671016949,-0.630490308557156],[0,0,0,0],[8.999999E+09,8.999999E+09,8.999999E+09,8.999999E+09,8.999999E+09,8.999999E+09]];
    LOCAL CONST Robtarget Tr_meulage_motif_1_292 := [[-23.640236328125,56.3248203125,37.019375],[0.325394831809823,-0.323189731818736,0.626217671016949,-0.630490308557156],[0,0,0,0],[8.999999E+09,8.999999E+09,8.999999E+09,8.999999E+09,8.999999E+09,8.999999E+09]];
    LOCAL CONST Robtarget Tr_meulage_motif_1_293 := [[-23.100931640625,57.1669296875,37.01937109375],[0.325394831809823,-0.323189731818736,0.626217671016949,-0.630490308557156],[0,0,0,0],[8.999999E+09,8.999999E+09,8.999999E+09,8.999999E+09,8.999999E+09,8.999999E+09]];
    LOCAL CONST Robtarget Tr_meulage_motif_1_294 := [[-22.561626953125,58.0090390625,37.01936328125],[0.325394831809823,-0.323189731818736,0.626217671016949,-0.630490308557156],[0,0,0,0],[8.999999E+09,8.999999E+09,8.999999E+09,8.999999E+09,8.999999E+09,8.999999E+09]];

